// SIMATIC STEP 7 (V5.x) project zhao2017
// CPU: CPU 315-2 DP
// station: Hardware
// station: SIMATIC 300(1)
// station: P_ADR_BUS
// program: S7 Program(1)

SYMBOL_TABLE
"F1_DATA"	DB 1	DB 1
"F2_DATA"	DB 2	DB 2
"DI/DO测试程序"	FC 31	FC 31
"AI/AO测试程序"	FC 32	FC 32
"端子控制"	FC 41	FC 41
"PPO1通讯子程序"	FC 60	FC 60
"单机启停控制"	FC 71	FC 71
"加减速子程序"	FC 72	FC 72
"同步逻辑程序"	FC 81	FC 81
"单机速度程序"	FC 82	FC 82
"同步速度程序"	FC 83	FC 83
"显示与通讯程序"	FC 84	FC 84
"S1_run"	I 0.0	BOOL	// M150.0
"S1_stop"	I 0.1	BOOL	// M150.1
"S1_inc"	I 0.2	BOOL	// M150.2
"S1_dec"	I 0.3	BOOL	// M150.3
"S4_run"	I 1.4	BOOL	// M150.6
"S4_stop"	I 1.5	BOOL	// M150.7
"S4_inc"	I 1.6	BOOL	// M151.0
"S4_dec"	I 1.7	BOOL	// M151.1
"S5_run"	I 4.0	BOOL	// M151.4
"S5_stop"	I 4.1	BOOL	// M151.5
"F1"	I 6.0	BOOL	// M151.6
"F2"	I 6.1	BOOL	// M151.7
"zeroadj"	I 6.6	BOOL
"maxadj"	I 6.7	BOOL
"pulse"	M 20.0	BOOL
"T1S"	M 20.1	BOOL
"S1_running"	M 70.0	BOOL
"S4_running"	M 70.1	BOOL
"S1_Run_Mode"	M 70.2	BOOL
"S4_Run_Mode"	M 70.5	BOOL
"S1_P1"	M 80.0	BOOL
"S1_P2"	M 80.1	BOOL
"S1_P3"	M 80.2	BOOL
"S1_P4"	M 80.3	BOOL
"S1_P5"	M 80.4	BOOL
"S1_P6"	M 80.5	BOOL
"S1_P7"	M 80.6	BOOL
"S4_P1"	M 81.0	BOOL
"S4_P2"	M 81.1	BOOL
"S4_P3"	M 81.2	BOOL
"S4_P4"	M 81.3	BOOL
"S4_P5"	M 81.4	BOOL
"S4_P6"	M 81.5	BOOL
"S4_P7"	M 81.6	BOOL
"S4_P8"	M 81.7	BOOL
"S1_P8"	M 82.0	BOOL
"S1_stoped"	M 82.2	BOOL
"S4_stoped"	M 82.3	BOOL
"S1_running_order"	M 83.0	BOOL
"S4_running_order"	M 83.1	BOOL
"T50ms"	M 200.0	BOOL
"S1_running_p"	M 200.1	BOOL
"T 50MS"	M 200.2	BOOL
"S4_running_p"	M 200.3	BOOL
"S1_speed"	PQW 304	WORD
"S5_speed"	PQW 308	WORD
"S4_speed"	PQW 310	WORD
"S5_1speed"	PQW 320	WORD
"S1_run_lamp"	Q 8.0	BOOL	// M150.4
"S1_stop_lamp"	Q 8.1	BOOL	// M150.5
"S4_run_lamp"	Q 8.6	BOOL	// M151.2
"S4_stop_lamp"	Q 8.7	BOOL	// M151.3
"DPRD_DAT"	SFC 14	SFC 14	// Read Consistent Data of a Standard DP Slave
"DPWR_DAT"	SFC 15	SFC 15	// Write Consistent Data to a Standard DP Slave
END_SYMBOL_TABLE

FUNCTION "DI/DO测试程序" : VOID	// FC 31
VERSION : 0.1
BEGIN
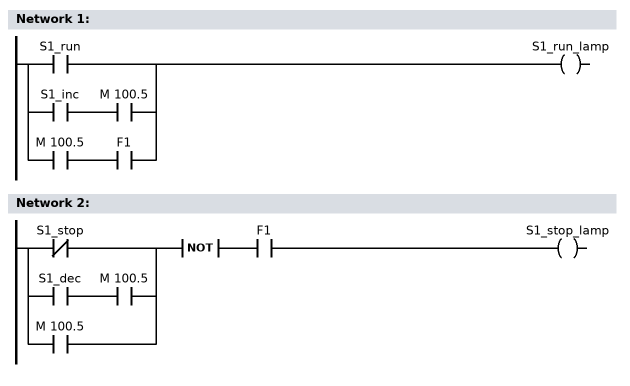
NETWORK
TITLE =
      O     "S1_run";
      O;
      A     "S1_inc";
      A     M 100.5;
      O;
      A     M 100.5;
      A     "F1";
      =     "S1_run_lamp";
NETWORK
TITLE =
      ON    "S1_stop";
      O;
      A     "S1_dec";
      A     M 100.5;
      O;
      A     M 100.5;
      NOT;
      A     "F1";
      =     "S1_stop_lamp";
END_FUNCTION

FUNCTION "AI/AO测试程序" : VOID	// FC 32
VERSION : 0.1
BEGIN
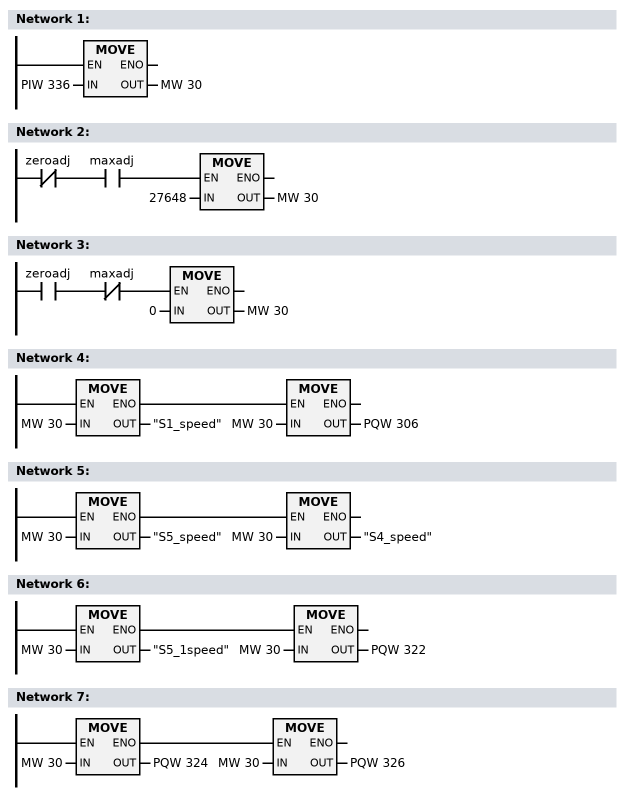
NETWORK
TITLE =
      L     PIW 336;
      T     MW 30;
      NOP   0;
NETWORK
TITLE =
      AN    "zeroadj";
      A     "maxadj";
      JNB   _001;
      L     27648;
      T     MW 30;
_001: NOP   0;
NETWORK
TITLE =
      A     "zeroadj";
      AN    "maxadj";
      JNB   _002;
      L     0;
      T     MW 30;
_002: NOP   0;
NETWORK
TITLE =
      A(;
      L     MW 30;
      T     "S1_speed";
      SET;
      SAVE;
      CLR;
      A     BR;
      );
      JNB   _003;
      L     MW 30;
      T     PQW 306;
_003: NOP   0;
NETWORK
TITLE =
      A(;
      L     MW 30;
      T     "S5_speed";
      SET;
      SAVE;
      CLR;
      A     BR;
      );
      JNB   _004;
      L     MW 30;
      T     "S4_speed";
_004: NOP   0;
NETWORK
TITLE =
      A(;
      L     MW 30;
      T     "S5_1speed";
      SET;
      SAVE;
      CLR;
      A     BR;
      );
      JNB   _005;
      L     MW 30;
      T     PQW 322;
_005: NOP   0;
NETWORK
TITLE =
      A(;
      L     MW 30;
      T     PQW 324;
      SET;
      SAVE;
      CLR;
      A     BR;
      );
      JNB   _006;
      L     MW 30;
      T     PQW 326;
_006: NOP   0;
NETWORK
TITLE =
END_FUNCTION

FUNCTION "端子控制" : VOID	// FC 41
VERSION : 0.1
BEGIN
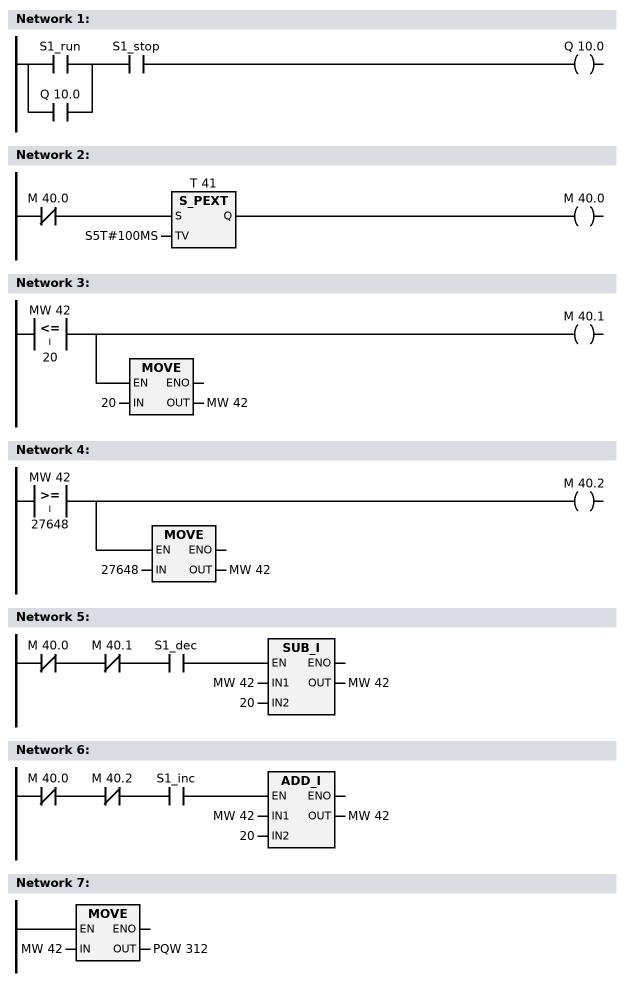
NETWORK
TITLE =
      A(;
      O     "S1_run";
      O     Q 10.0;
      );
      A     "S1_stop";
      =     Q 10.0;
NETWORK
TITLE =
      AN    M 40.0;
      L     S5T#100MS;
      SE    T 41;
      NOP   0;
      NOP   0;
      NOP   0;
      A     T 41;
      =     M 40.0;
NETWORK
TITLE =
      L     MW 42;
      L     20;
      <=I;
      =     L 0.0;
      A     L 0.0;
      BLD   102;
      =     M 40.1;
      A     L 0.0;
      JNB   _001;
      L     20;
      T     MW 42;
_001: NOP   0;
NETWORK
TITLE =
      L     MW 42;
      L     27648;
      >=I;
      =     L 0.0;
      A     L 0.0;
      BLD   102;
      =     M 40.2;
      A     L 0.0;
      JNB   _002;
      L     27648;
      T     MW 42;
_002: NOP   0;
NETWORK
TITLE =
      AN    M 40.0;
      AN    M 40.1;
      A     "S1_dec";
      JNB   _003;
      L     MW 42;
      L     20;
      -I;
      T     MW 42;
_003: NOP   0;
NETWORK
TITLE =
      AN    M 40.0;
      AN    M 40.2;
      A     "S1_inc";
      JNB   _004;
      L     MW 42;
      L     20;
      +I;
      T     MW 42;
_004: NOP   0;
NETWORK
TITLE =
      L     MW 42;
      T     PQW 312;
      NOP   0;
NETWORK
TITLE =
END_FUNCTION

FUNCTION "PPO1通讯子程序" : VOID	// FC 60
VERSION : 0.1
VAR_INPUT
  pkw1 : WORD ;
  pkw2 : WORD ;
  pkw3 : WORD ;
  pkw4 : WORD ;
  pzd1 : WORD ;
  pzd2 : INT ;
  pkw_I_addr : WORD ;
  pkw_Q_addr : WORD ;
  pzd_I_addr : WORD ;
  pzd_Q_addr : WORD ;
END_VAR
VAR_OUTPUT
  pkw1_ret : WORD ;
  pkw2_ret : WORD ;
  pkw3_ret : WORD ;
  pkw4_ret : WORD ;
  pzd1_ret : WORD ;
  pzd2_ret : WORD ;
  err : BOOL ;
END_VAR
VAR_TEMP
  pkw : STRUCT
   w1 : WORD ;
   w2 : WORD ;
   w3 : WORD ;
   w4 : WORD ;
  END_STRUCT ;
  pzd : STRUCT
   w1 : WORD ;
   w2 : WORD ;
  END_STRUCT ;
  pkw_RD : STRUCT
   w1 : WORD ;
   w2 : WORD ;
   w3 : WORD ;
   w4 : WORD ;
  END_STRUCT ;
  pzd_RD : STRUCT
   w1 : WORD ;
   w2 : WORD ;
  END_STRUCT ;
  tt : STRUCT
   w1 : INT ;
   w2 : INT ;
   w3 : INT ;
   w4 : INT ;
  END_STRUCT ;
END_VAR
BEGIN
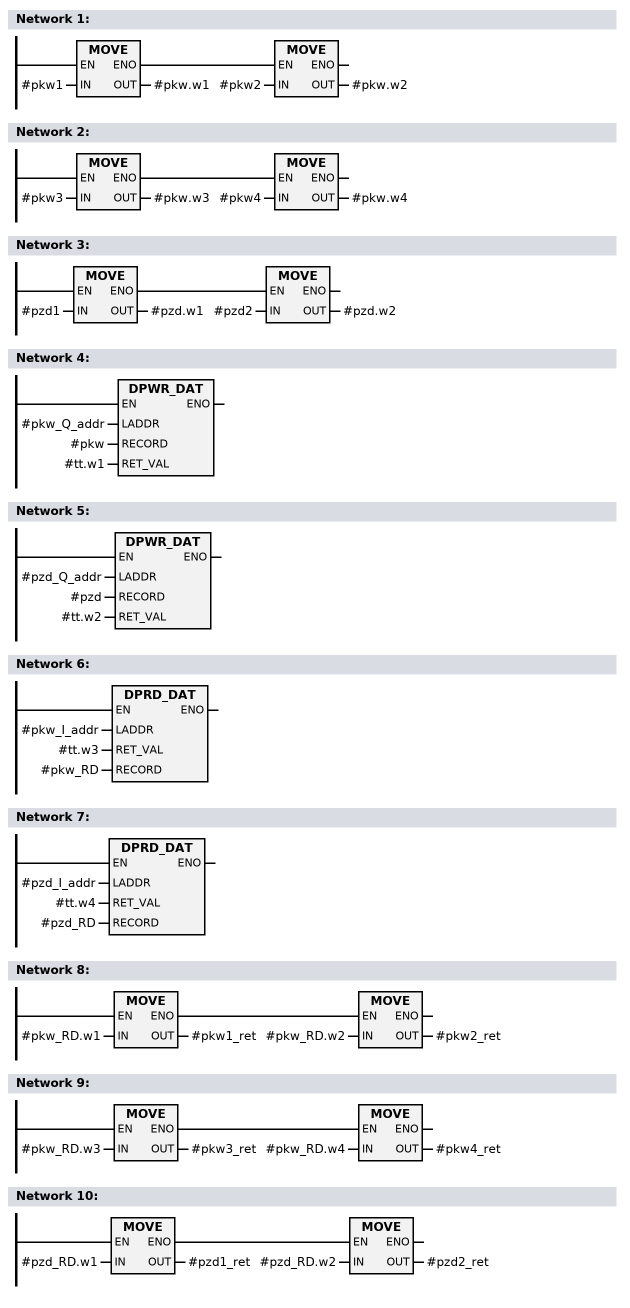
NETWORK
TITLE =
//将pkw1、pkw2数据放入变量组
      A(;
      L     #pkw1;
      T     #pkw.w1;
      SET;
      SAVE;
      CLR;
      A     BR;
      );
      JNB   _001;
      L     #pkw2;
      T     #pkw.w2;
_001: NOP   0;
NETWORK
TITLE =
//将pkw3、pkw4数据放入变量组
      A(;
      L     #pkw3;
      T     #pkw.w3;
      SET;
      SAVE;
      CLR;
      A     BR;
      );
      JNB   _002;
      L     #pkw4;
      T     #pkw.w4;
_002: NOP   0;
NETWORK
TITLE =
//将pzd数据放入变量组
      A(;
      L     #pzd1;
      T     #pzd.w1;
      SET;
      SAVE;
      CLR;
      A     BR;
      );
      JNB   _003;
      L     #pzd2;
      T     #pzd.w2;
_003: NOP   0;
NETWORK
TITLE =
//将pkw数据输出
      CALL  "DPWR_DAT" (
           LADDR                    := #pkw_Q_addr,
           RECORD                   := #pkw,
           RET_VAL                  := #tt.w1);
      NOP   0;
NETWORK
TITLE =
//将pzd数据输出
      CALL  "DPWR_DAT" (
           LADDR                    := #pzd_Q_addr,
           RECORD                   := #pzd,
           RET_VAL                  := #tt.w2);
      NOP   0;
NETWORK
TITLE =
//将pkw响应数据读入
      CALL  "DPRD_DAT" (
           LADDR                    := #pkw_I_addr,
           RET_VAL                  := #tt.w3,
           RECORD                   := #pkw_RD);
      NOP   0;
NETWORK
TITLE =
//将pzd响应数据读入
      CALL  "DPRD_DAT" (
           LADDR                    := #pzd_I_addr,
           RET_VAL                  := #tt.w4,
           RECORD                   := #pzd_RD);
      NOP   0;
NETWORK
TITLE =
//把读入的数据放入PKW响应数据区相应位置
      A(;
      L     #pkw_RD.w1;
      T     #pkw1_ret;
      SET;
      SAVE;
      CLR;
      A     BR;
      );
      JNB   _004;
      L     #pkw_RD.w2;
      T     #pkw2_ret;
_004: NOP   0;
NETWORK
TITLE =
//把读入的数据放入PKW响应数据区相应位置
      A(;
      L     #pkw_RD.w3;
      T     #pkw3_ret;
      SET;
      SAVE;
      CLR;
      A     BR;
      );
      JNB   _005;
      L     #pkw_RD.w4;
      T     #pkw4_ret;
_005: NOP   0;
NETWORK
TITLE =
//把读入的数据放入PZD响应数据区相应位置
      A(;
      L     #pzd_RD.w1;
      T     #pzd1_ret;
      SET;
      SAVE;
      CLR;
      A     BR;
      );
      JNB   _006;
      L     #pzd_RD.w2;
      T     #pzd2_ret;
_006: NOP   0;
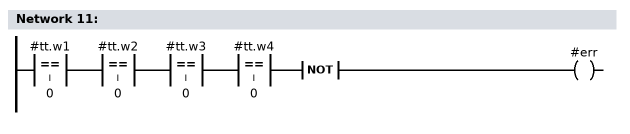
NETWORK
TITLE =
      A(;
      L     #tt.w1;
      L     0;
      ==I;
      );
      A(;
      L     #tt.w2;
      L     0;
      ==I;
      );
      A(;
      L     #tt.w3;
      L     0;
      ==I;
      );
      A(;
      L     #tt.w4;
      L     0;
      ==I;
      );
      NOT;
      =     #err;
END_FUNCTION

FUNCTION "单机启停控制" : VOID	// FC 71
VERSION : 0.1
BEGIN
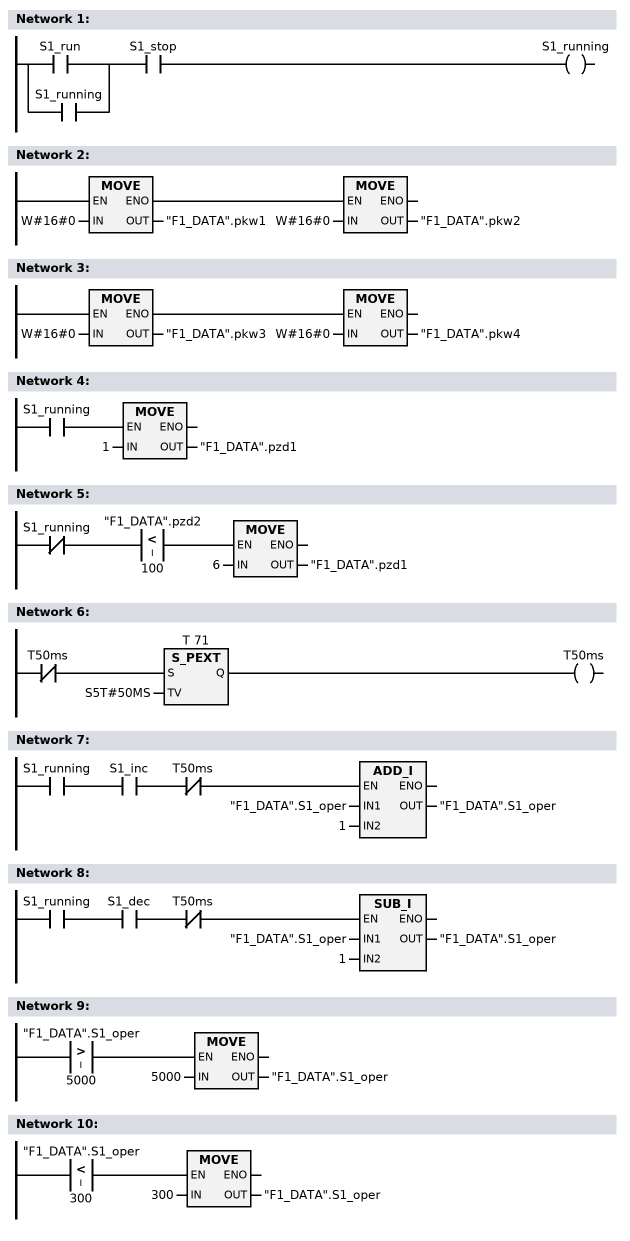
NETWORK
TITLE =
      A(;
      O     "S1_run";
      O     "S1_running";
      );
      A     "S1_stop";
      =     "S1_running";
NETWORK
TITLE =
      A(;
      L     W#16#0;
      T     "F1_DATA".pkw1;
      SET;
      SAVE;
      CLR;
      A     BR;
      );
      JNB   _001;
      L     W#16#0;
      T     "F1_DATA".pkw2;
_001: NOP   0;
NETWORK
TITLE =
      A(;
      L     W#16#0;
      T     "F1_DATA".pkw3;
      SET;
      SAVE;
      CLR;
      A     BR;
      );
      JNB   _002;
      L     W#16#0;
      T     "F1_DATA".pkw4;
_002: NOP   0;
NETWORK
TITLE =
      A     "S1_running";
      JNB   _003;
      L     1;
      T     "F1_DATA".pzd1;
_003: NOP   0;
NETWORK
TITLE =
      AN    "S1_running";
      A(;
      L     "F1_DATA".pzd2;
      L     100;
      <I;
      );
      JNB   _004;
      L     6;
      T     "F1_DATA".pzd1;
_004: NOP   0;
NETWORK
TITLE =
      AN    "T50ms";
      L     S5T#50MS;
      SE    T 71;
      NOP   0;
      NOP   0;
      NOP   0;
      A     T 71;
      =     "T50ms";
NETWORK
TITLE =
      A     "S1_running";
      A     "S1_inc";
      AN    "T50ms";
      JNB   _005;
      L     "F1_DATA".S1_oper;
      L     1;
      +I;
      T     "F1_DATA".S1_oper;
_005: NOP   0;
NETWORK
TITLE =
      A     "S1_running";
      A     "S1_dec";
      AN    "T50ms";
      JNB   _006;
      L     "F1_DATA".S1_oper;
      L     1;
      -I;
      T     "F1_DATA".S1_oper;
_006: NOP   0;
NETWORK
TITLE =
      A(;
      L     "F1_DATA".S1_oper;
      L     5000;
      >I;
      );
      JNB   _007;
      L     5000;
      T     "F1_DATA".S1_oper;
_007: NOP   0;
NETWORK
TITLE =
      A(;
      L     "F1_DATA".S1_oper;
      L     300;
      <I;
      );
      JNB   _008;
      L     300;
      T     "F1_DATA".S1_oper;
_008: NOP   0;
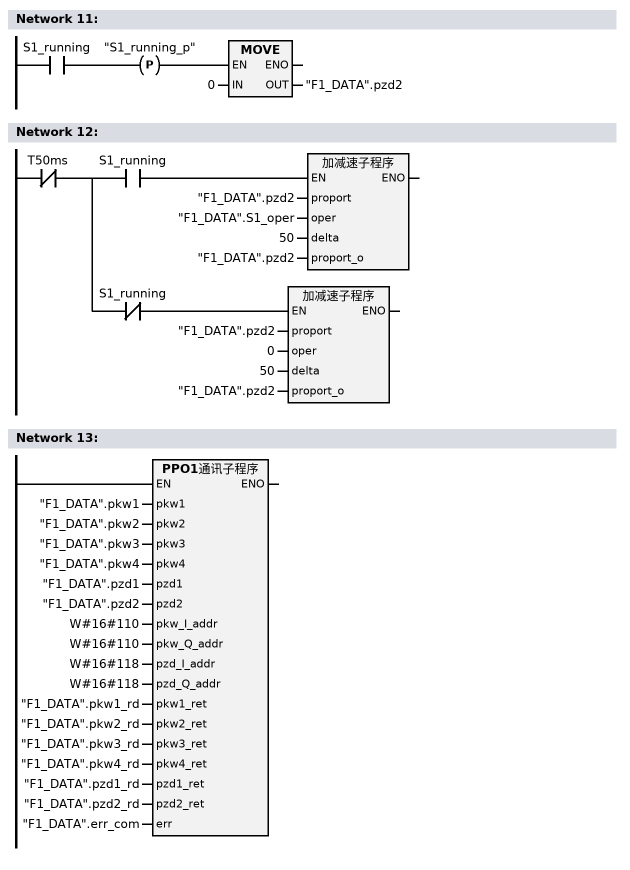
NETWORK
TITLE =
      A     "S1_running";
      FP    "S1_running_p";
      JNB   _009;
      L     0;
      T     "F1_DATA".pzd2;
_009: NOP   0;
NETWORK
TITLE =
      AN    "T50ms";
      =     L 0.0;
      A     L 0.0;
      A     "S1_running";
      JNB   _00a;
      CALL  "加减速子程序" (
           proport                  := "F1_DATA".pzd2,
           oper                     := "F1_DATA".S1_oper,
           delta                    := 50,
           proport_o                := "F1_DATA".pzd2);
_00a: NOP   0;
      A     L 0.0;
      AN    "S1_running";
      JNB   _00b;
      CALL  "加减速子程序" (
           proport                  := "F1_DATA".pzd2,
           oper                     := 0,
           delta                    := 50,
           proport_o                := "F1_DATA".pzd2);
_00b: NOP   0;
NETWORK
TITLE =
      CALL  "PPO1通讯子程序" (
           pkw1                     := "F1_DATA".pkw1,
           pkw2                     := "F1_DATA".pkw2,
           pkw3                     := "F1_DATA".pkw3,
           pkw4                     := "F1_DATA".pkw4,
           pzd1                     := "F1_DATA".pzd1,
           pzd2                     := "F1_DATA".pzd2,
           pkw_I_addr               := W#16#110,
           pkw_Q_addr               := W#16#110,
           pzd_I_addr               := W#16#118,
           pzd_Q_addr               := W#16#118,
           pkw1_ret                 := "F1_DATA".pkw1_rd,
           pkw2_ret                 := "F1_DATA".pkw2_rd,
           pkw3_ret                 := "F1_DATA".pkw3_rd,
           pkw4_ret                 := "F1_DATA".pkw4_rd,
           pzd1_ret                 := "F1_DATA".pzd1_rd,
           pzd2_ret                 := "F1_DATA".pzd2_rd,
           err                      := "F1_DATA".err_com);
      NOP   0;
END_FUNCTION

FUNCTION "加减速子程序" : VOID	// FC 72
VERSION : 0.1
VAR_INPUT
  proport : INT ;
  oper : INT ;
  delta : INT ;
END_VAR
VAR_OUTPUT
  proport_o : INT ;
END_VAR
VAR_TEMP
  temp1 : BOOL ;
  temp2 : INT ;
END_VAR
BEGIN
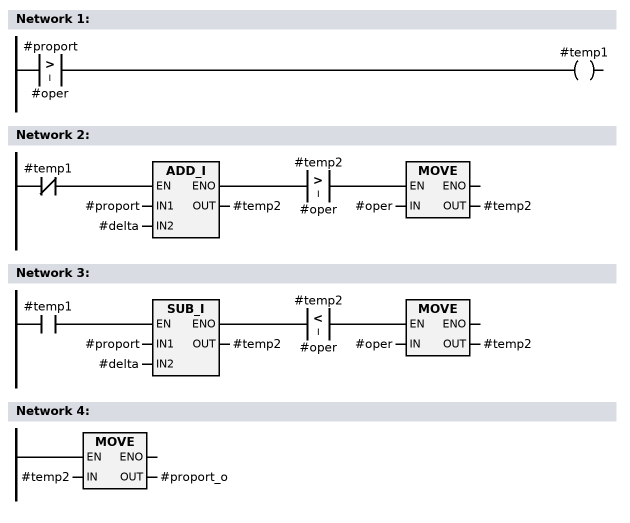
NETWORK
TITLE =
      L     #proport;
      L     #oper;
      >I;
      =     #temp1;
NETWORK
TITLE =
      A(;
      AN    #temp1;
      JNB   _001;
      L     #proport;
      L     #delta;
      +I;
      T     #temp2;
      AN    OV;
      SAVE;
      CLR;
_001: A     BR;
      );
      A(;
      L     #temp2;
      L     #oper;
      >I;
      );
      JNB   _002;
      L     #oper;
      T     #temp2;
_002: NOP   0;
NETWORK
TITLE =
      A(;
      A     #temp1;
      JNB   _003;
      L     #proport;
      L     #delta;
      -I;
      T     #temp2;
      AN    OV;
      SAVE;
      CLR;
_003: A     BR;
      );
      A(;
      L     #temp2;
      L     #oper;
      <I;
      );
      JNB   _004;
      L     #oper;
      T     #temp2;
_004: NOP   0;
NETWORK
TITLE =
      L     #temp2;
      T     #proport_o;
      NOP   0;
END_FUNCTION

FUNCTION "同步逻辑程序" : VOID	// FC 81
VERSION : 0.1
BEGIN
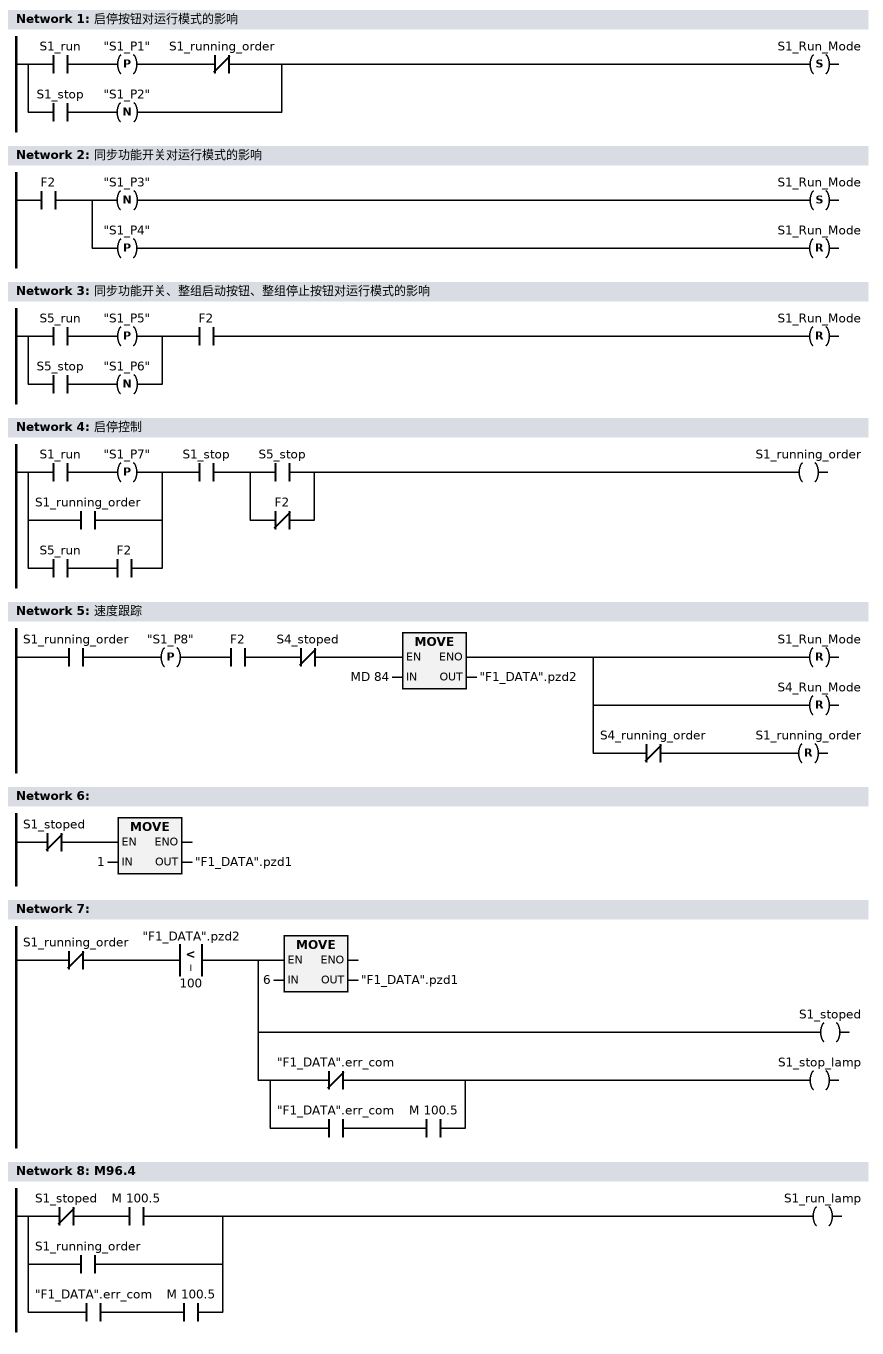
NETWORK
TITLE = 启停按钮对运行模式的影响
//Run_Mode=1表示单机运行，Run_Mode=0表示同步运行
      A     "S1_run";
      FP    "S1_P1";
      AN    "S1_running_order";
      O(;
      A     "S1_stop";
      FN    "S1_P2";
      );
      S     "S1_Run_Mode";
NETWORK
TITLE = 同步功能开关对运行模式的影响
//Run_Mode=1表示单机运行，Run_Mode=0表示同步运行
      A     "F2";
      =     L 0.0;
      A     L 0.0;
      FN    "S1_P3";
      S     "S1_Run_Mode";
      A     L 0.0;
      FP    "S1_P4";
      R     "S1_Run_Mode";
NETWORK
TITLE = 同步功能开关、整组启动按钮、整组停止按钮对运行模式的影响
//Run_Mode=1表示单机运行，Run_Mode=0表示同步运行
//“S3启动”（I1.0）为整组启动按钮，“S3停止”（I1.1）为整组停止按钮。
      A(;
      A     "S5_run";
      FP    "S1_P5";
      O(;
      A     "S5_stop";
      FN    "S1_P6";
      );
      );
      A     "F2";
      R     "S1_Run_Mode";
NETWORK
TITLE = 启停控制
//“F2”（I6.1）为同步功能开关，即I6.1=0时，两台变频器单机运行，I6.1=1时，两台变频
//器同步运行
      A(;
      A     "S1_run";
      FP    "S1_P7";
      O     "S1_running_order";
      O;
      A     "S5_run";
      A     "F2";
      );
      A     "S1_stop";
      A(;
      O     "S5_stop";
      ON    "F2";
      );
      =     "S1_running_order";
NETWORK
TITLE = 速度跟踪
//Run_Mode=1表示单机运行，Run_Mode=0表示同步运行
      A     "S1_running_order";
      FP    "S1_P8";
      A     "F2";
      AN    "S4_stoped";
      JNB   _001;
      L     MD 84;
      T     "F1_DATA".pzd2;
      SET;
      SAVE;
      CLR;
_001: A     BR;
      =     L 0.0;
      A     L 0.0;
      BLD   102;
      R     "S1_Run_Mode";
      A     L 0.0;
      BLD   102;
      R     "S4_Run_Mode";
      A     L 0.0;
      AN    "S4_running_order";
      R     "S1_running_order";
NETWORK
TITLE =
      AN    "S1_stoped";
      JNB   _002;
      L     1;
      T     "F1_DATA".pzd1;
_002: NOP   0;
NETWORK
TITLE =
      AN    "S1_running_order";
      A(;
      L     "F1_DATA".pzd2;
      L     100;
      <I;
      );
      =     L 0.0;
      A     L 0.0;
      JNB   _003;
      L     6;
      T     "F1_DATA".pzd1;
_003: NOP   0;
      A     L 0.0;
      BLD   102;
      =     "S1_stoped";
      A     L 0.0;
      A(;
      ON    "F1_DATA".err_com;
      O;
      A     "F1_DATA".err_com;
      A     M 100.5;
      );
      =     "S1_stop_lamp";
NETWORK
TITLE = M96.4
      AN    "S1_stoped";
      A     M 100.5;
      O     "S1_running_order";
      O;
      A     "F1_DATA".err_com;
      A     M 100.5;
      =     "S1_run_lamp";
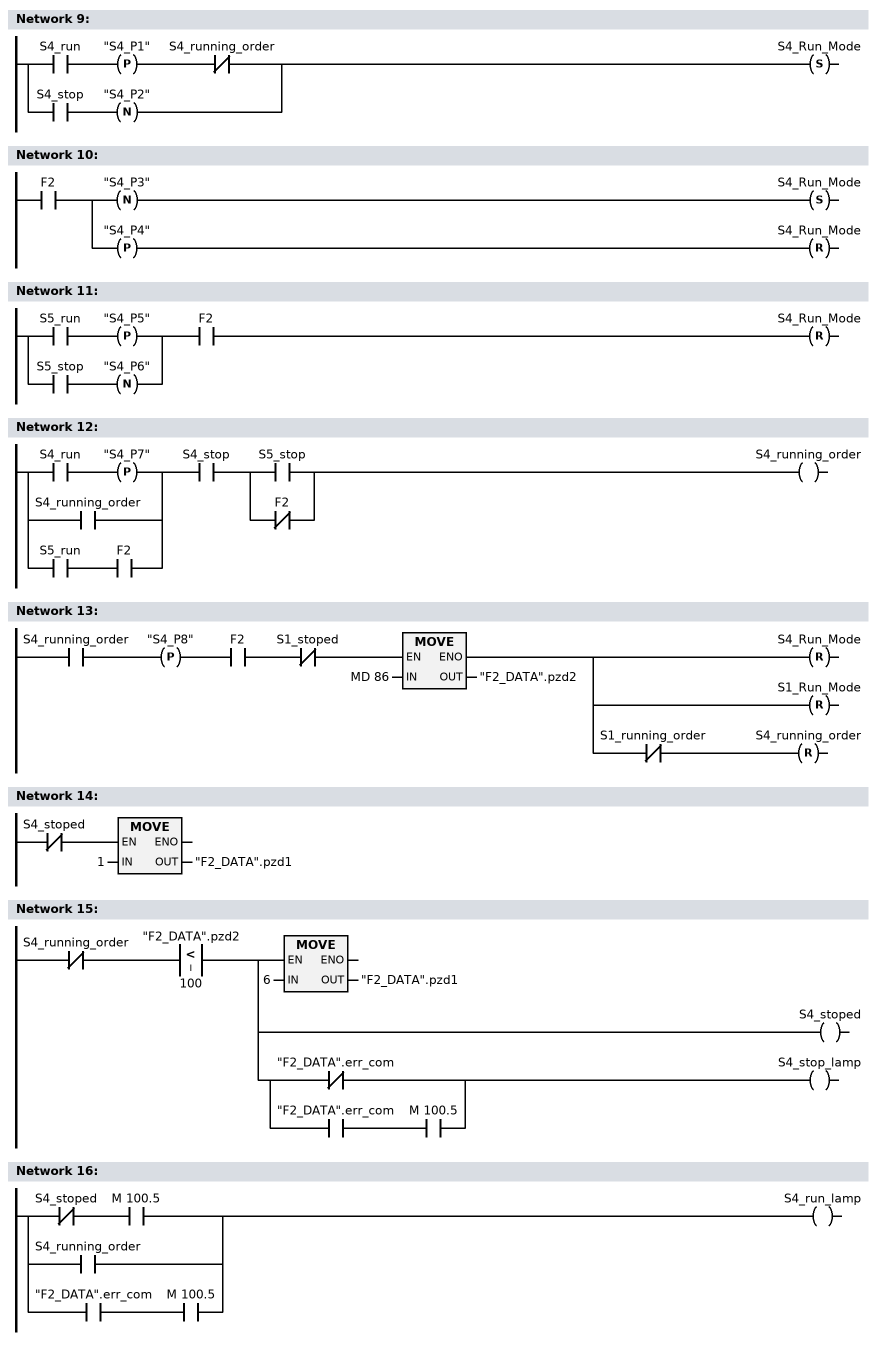
NETWORK
TITLE =
      A     "S4_run";
      FP    "S4_P1";
      AN    "S4_running_order";
      O(;
      A     "S4_stop";
      FN    "S4_P2";
      );
      S     "S4_Run_Mode";
NETWORK
TITLE =
      A     "F2";
      =     L 0.0;
      A     L 0.0;
      FN    "S4_P3";
      S     "S4_Run_Mode";
      A     L 0.0;
      FP    "S4_P4";
      R     "S4_Run_Mode";
NETWORK
TITLE =
      A(;
      A     "S5_run";
      FP    "S4_P5";
      O(;
      A     "S5_stop";
      FN    "S4_P6";
      );
      );
      A     "F2";
      R     "S4_Run_Mode";
NETWORK
TITLE =
      A(;
      A     "S4_run";
      FP    "S4_P7";
      O     "S4_running_order";
      O;
      A     "S5_run";
      A     "F2";
      );
      A     "S4_stop";
      A(;
      O     "S5_stop";
      ON    "F2";
      );
      =     "S4_running_order";
NETWORK
TITLE =
      A     "S4_running_order";
      FP    "S4_P8";
      A     "F2";
      AN    "S1_stoped";
      JNB   _004;
      L     MD 86;
      T     "F2_DATA".pzd2;
      SET;
      SAVE;
      CLR;
_004: A     BR;
      =     L 0.0;
      A     L 0.0;
      BLD   102;
      R     "S4_Run_Mode";
      A     L 0.0;
      BLD   102;
      R     "S1_Run_Mode";
      A     L 0.0;
      AN    "S1_running_order";
      R     "S4_running_order";
NETWORK
TITLE =
      AN    "S4_stoped";
      JNB   _005;
      L     1;
      T     "F2_DATA".pzd1;
_005: NOP   0;
NETWORK
TITLE =
      AN    "S4_running_order";
      A(;
      L     "F2_DATA".pzd2;
      L     100;
      <I;
      );
      =     L 0.0;
      A     L 0.0;
      JNB   _006;
      L     6;
      T     "F2_DATA".pzd1;
_006: NOP   0;
      A     L 0.0;
      BLD   102;
      =     "S4_stoped";
      A     L 0.0;
      A(;
      ON    "F2_DATA".err_com;
      O;
      A     "F2_DATA".err_com;
      A     M 100.5;
      );
      =     "S4_stop_lamp";
NETWORK
TITLE =
      AN    "S4_stoped";
      A     M 100.5;
      O     "S4_running_order";
      O;
      A     "F2_DATA".err_com;
      A     M 100.5;
      =     "S4_run_lamp";
END_FUNCTION

FUNCTION "单机速度程序" : VOID	// FC 82
VERSION : 0.1
VAR_TEMP
  S1_di_su : INT ;
  S2_di_su : INT ;
END_VAR
BEGIN
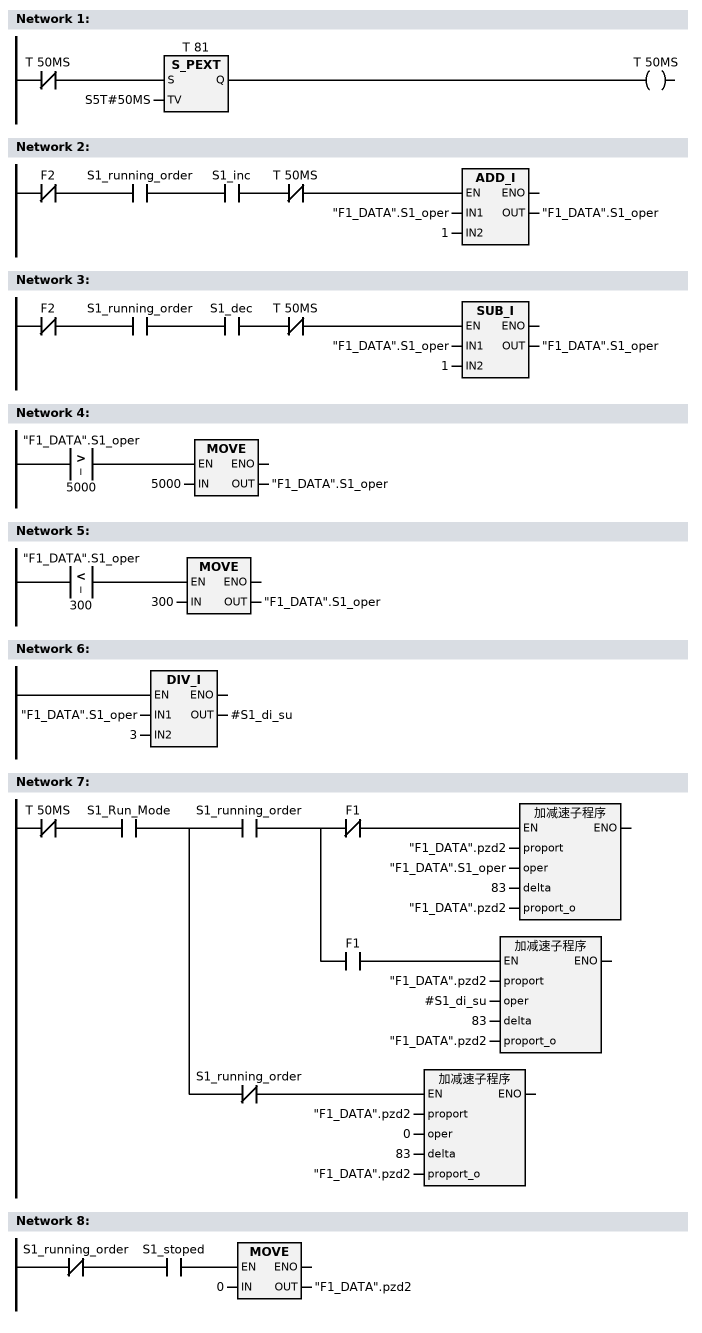
NETWORK
TITLE =
      AN    "T 50MS";
      L     S5T#50MS;
      SE    T 81;
      NOP   0;
      NOP   0;
      NOP   0;
      A     T 81;
      =     "T 50MS";
NETWORK
TITLE =
      AN    "F2";
      A     "S1_running_order";
      A     "S1_inc";
      AN    "T 50MS";
      JNB   _001;
      L     "F1_DATA".S1_oper;
      L     1;
      +I;
      T     "F1_DATA".S1_oper;
_001: NOP   0;
NETWORK
TITLE =
      AN    "F2";
      A     "S1_running_order";
      A     "S1_dec";
      AN    "T 50MS";
      JNB   _002;
      L     "F1_DATA".S1_oper;
      L     1;
      -I;
      T     "F1_DATA".S1_oper;
_002: NOP   0;
NETWORK
TITLE =
      A(;
      L     "F1_DATA".S1_oper;
      L     5000;
      >I;
      );
      JNB   _003;
      L     5000;
      T     "F1_DATA".S1_oper;
_003: NOP   0;
NETWORK
TITLE =
      A(;
      L     "F1_DATA".S1_oper;
      L     300;
      <I;
      );
      JNB   _004;
      L     300;
      T     "F1_DATA".S1_oper;
_004: NOP   0;
NETWORK
TITLE =
      L     "F1_DATA".S1_oper;
      L     3;
      /I;
      T     #S1_di_su;
      NOP   0;
NETWORK
TITLE =
      AN    "T 50MS";
      A     "S1_Run_Mode";
      =     L 4.0;
      A     L 4.0;
      A     "S1_running_order";
      =     L 4.1;
      A     L 4.1;
      AN    "F1";
      JNB   _005;
      CALL  "加减速子程序" (
           proport                  := "F1_DATA".pzd2,
           oper                     := "F1_DATA".S1_oper,
           delta                    := 83,
           proport_o                := "F1_DATA".pzd2);
_005: NOP   0;
      A     L 4.1;
      A     "F1";
      JNB   _006;
      CALL  "加减速子程序" (
           proport                  := "F1_DATA".pzd2,
           oper                     := #S1_di_su,
           delta                    := 83,
           proport_o                := "F1_DATA".pzd2);
_006: NOP   0;
      A     L 4.0;
      AN    "S1_running_order";
      JNB   _007;
      CALL  "加减速子程序" (
           proport                  := "F1_DATA".pzd2,
           oper                     := 0,
           delta                    := 83,
           proport_o                := "F1_DATA".pzd2);
_007: NOP   0;
NETWORK
TITLE =
      AN    "S1_running_order";
      A     "S1_stoped";
      JNB   _008;
      L     0;
      T     "F1_DATA".pzd2;
_008: NOP   0;
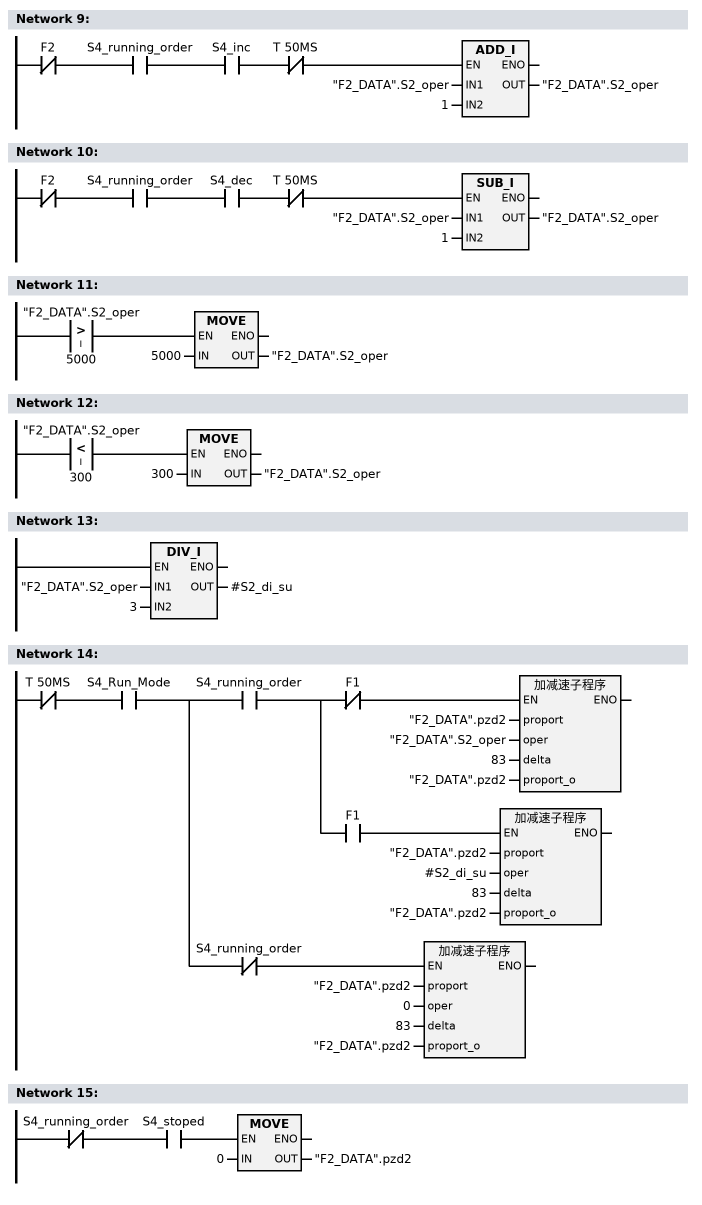
NETWORK
TITLE =
      AN    "F2";
      A     "S4_running_order";
      A     "S4_inc";
      AN    "T 50MS";
      JNB   _009;
      L     "F2_DATA".S2_oper;
      L     1;
      +I;
      T     "F2_DATA".S2_oper;
_009: NOP   0;
NETWORK
TITLE =
      AN    "F2";
      A     "S4_running_order";
      A     "S4_dec";
      AN    "T 50MS";
      JNB   _00a;
      L     "F2_DATA".S2_oper;
      L     1;
      -I;
      T     "F2_DATA".S2_oper;
_00a: NOP   0;
NETWORK
TITLE =
      A(;
      L     "F2_DATA".S2_oper;
      L     5000;
      >I;
      );
      JNB   _00b;
      L     5000;
      T     "F2_DATA".S2_oper;
_00b: NOP   0;
NETWORK
TITLE =
      A(;
      L     "F2_DATA".S2_oper;
      L     300;
      <I;
      );
      JNB   _00c;
      L     300;
      T     "F2_DATA".S2_oper;
_00c: NOP   0;
NETWORK
TITLE =
      L     "F2_DATA".S2_oper;
      L     3;
      /I;
      T     #S2_di_su;
      NOP   0;
NETWORK
TITLE =
      AN    "T 50MS";
      A     "S4_Run_Mode";
      =     L 4.0;
      A     L 4.0;
      A     "S4_running_order";
      =     L 4.1;
      A     L 4.1;
      AN    "F1";
      JNB   _00d;
      CALL  "加减速子程序" (
           proport                  := "F2_DATA".pzd2,
           oper                     := "F2_DATA".S2_oper,
           delta                    := 83,
           proport_o                := "F2_DATA".pzd2);
_00d: NOP   0;
      A     L 4.1;
      A     "F1";
      JNB   _00e;
      CALL  "加减速子程序" (
           proport                  := "F2_DATA".pzd2,
           oper                     := #S2_di_su,
           delta                    := 83,
           proport_o                := "F2_DATA".pzd2);
_00e: NOP   0;
      A     L 4.0;
      AN    "S4_running_order";
      JNB   _00f;
      CALL  "加减速子程序" (
           proport                  := "F2_DATA".pzd2,
           oper                     := 0,
           delta                    := 83,
           proport_o                := "F2_DATA".pzd2);
_00f: NOP   0;
NETWORK
TITLE =
      AN    "S4_running_order";
      A     "S4_stoped";
      JNB   _010;
      L     0;
      T     "F2_DATA".pzd2;
_010: NOP   0;
END_FUNCTION

FUNCTION "同步速度程序" : VOID	// FC 83
VERSION : 0.1
VAR_TEMP
  TEMP0 : DINT ;
  TEMP1 : REAL ;
  TEMP2 : DINT ;
  TEMP3 : REAL ;
  S1_di_su : INT ;
  S2_di_su : INT ;
END_VAR
BEGIN
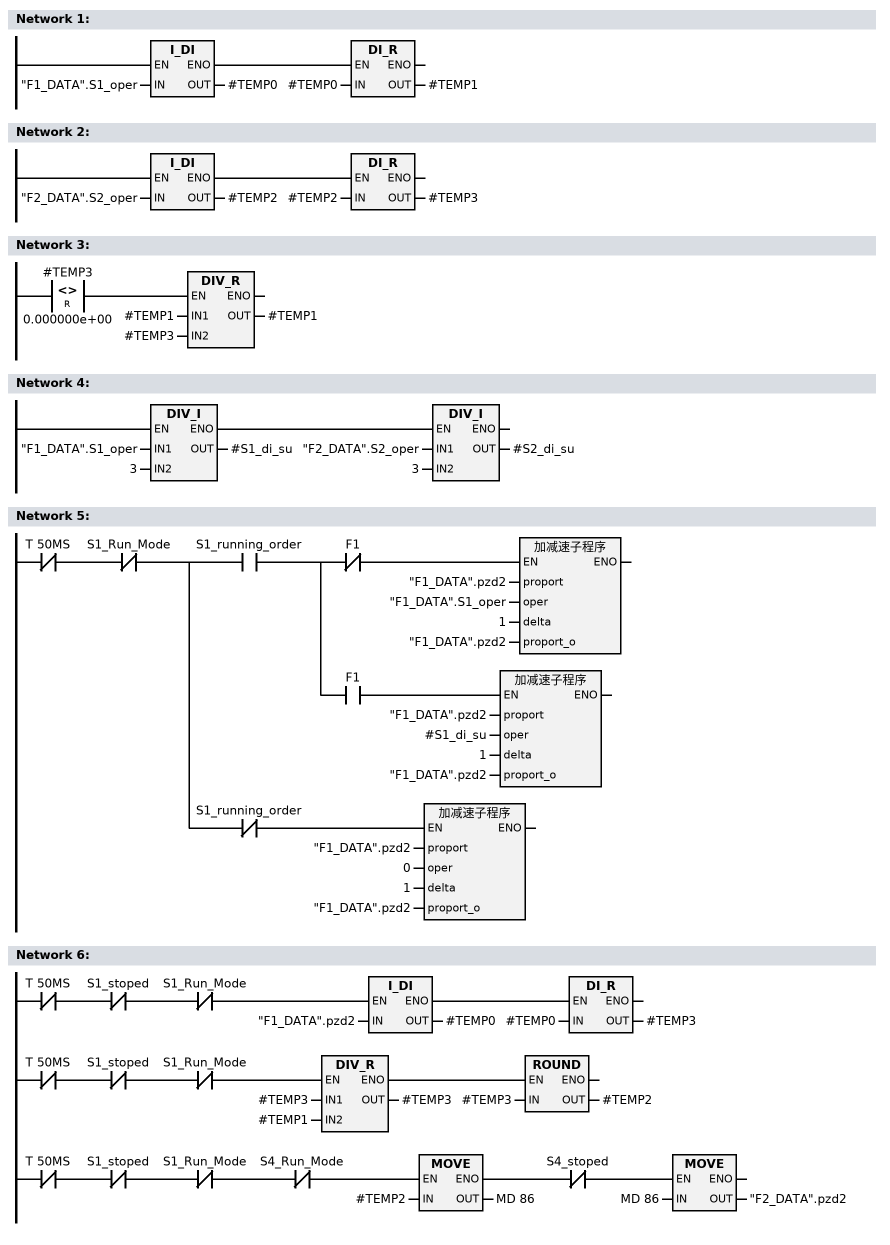
NETWORK
TITLE =
      A(;
      L     "F1_DATA".S1_oper;
      ITD;
      T     #TEMP0;
      SET;
      SAVE;
      CLR;
      A     BR;
      );
      JNB   _001;
      L     #TEMP0;
      DTR;
      T     #TEMP1;
_001: NOP   0;
NETWORK
TITLE =
      A(;
      L     "F2_DATA".S2_oper;
      ITD;
      T     #TEMP2;
      SET;
      SAVE;
      CLR;
      A     BR;
      );
      JNB   _002;
      L     #TEMP2;
      DTR;
      T     #TEMP3;
_002: NOP   0;
NETWORK
TITLE =
      A(;
      L     #TEMP3;
      L     0.000000e+00;
      <>R;
      );
      JNB   _003;
      L     #TEMP1;
      L     #TEMP3;
      /R;
      T     #TEMP1;
_003: NOP   0;
NETWORK
TITLE =
      A(;
      L     "F1_DATA".S1_oper;
      L     3;
      /I;
      T     #S1_di_su;
      AN    OV;
      SAVE;
      CLR;
      A     BR;
      );
      JNB   _004;
      L     "F2_DATA".S2_oper;
      L     3;
      /I;
      T     #S2_di_su;
_004: NOP   0;
NETWORK
TITLE =
      AN    "T 50MS";
      AN    "S1_Run_Mode";
      =     L 20.0;
      A     L 20.0;
      A     "S1_running_order";
      =     L 20.1;
      A     L 20.1;
      AN    "F1";
      JNB   _005;
      CALL  "加减速子程序" (
           proport                  := "F1_DATA".pzd2,
           oper                     := "F1_DATA".S1_oper,
           delta                    := 1,
           proport_o                := "F1_DATA".pzd2);
_005: NOP   0;
      A     L 20.1;
      A     "F1";
      JNB   _006;
      CALL  "加减速子程序" (
           proport                  := "F1_DATA".pzd2,
           oper                     := #S1_di_su,
           delta                    := 1,
           proport_o                := "F1_DATA".pzd2);
_006: NOP   0;
      A     L 20.0;
      AN    "S1_running_order";
      JNB   _007;
      CALL  "加减速子程序" (
           proport                  := "F1_DATA".pzd2,
           oper                     := 0,
           delta                    := 1,
           proport_o                := "F1_DATA".pzd2);
_007: NOP   0;
NETWORK
TITLE =
      AN    "T 50MS";
      AN    "S1_stoped";
      AN    "S1_Run_Mode";
      =     L 20.0;
      A(;
      A     L 20.0;
      JNB   _008;
      L     "F1_DATA".pzd2;
      ITD;
      T     #TEMP0;
      SET;
      SAVE;
      CLR;
_008: A     BR;
      );
      JNB   _009;
      L     #TEMP0;
      DTR;
      T     #TEMP3;
_009: NOP   0;
      A(;
      A     L 20.0;
      JNB   _00a;
      L     #TEMP3;
      L     #TEMP1;
      /R;
      T     #TEMP3;
      AN    OV;
      SAVE;
      CLR;
_00a: A     BR;
      );
      JNB   _00b;
      L     #TEMP3;
      RND;
      T     #TEMP2;
_00b: NOP   0;
      A(;
      A     L 20.0;
      AN    "S4_Run_Mode";
      JNB   _00c;
      L     #TEMP2;
      T     MD 86;
      SET;
      SAVE;
      CLR;
_00c: A     BR;
      );
      AN    "S4_stoped";
      JNB   _00d;
      L     MD 86;
      T     "F2_DATA".pzd2;
_00d: NOP   0;
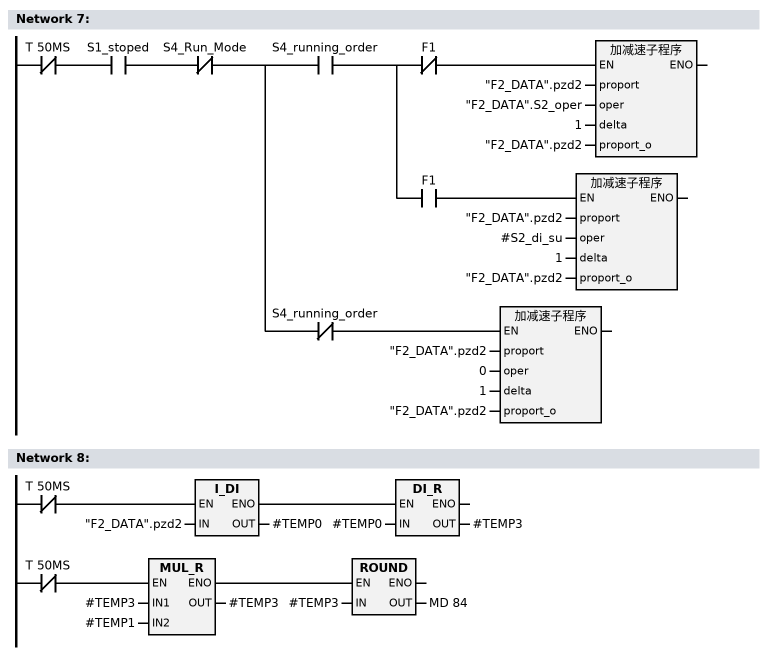
NETWORK
TITLE =
      AN    "T 50MS";
      A     "S1_stoped";
      AN    "S4_Run_Mode";
      =     L 20.0;
      A     L 20.0;
      A     "S4_running_order";
      =     L 20.1;
      A     L 20.1;
      AN    "F1";
      JNB   _00e;
      CALL  "加减速子程序" (
           proport                  := "F2_DATA".pzd2,
           oper                     := "F2_DATA".S2_oper,
           delta                    := 1,
           proport_o                := "F2_DATA".pzd2);
_00e: NOP   0;
      A     L 20.1;
      A     "F1";
      JNB   _00f;
      CALL  "加减速子程序" (
           proport                  := "F2_DATA".pzd2,
           oper                     := #S2_di_su,
           delta                    := 1,
           proport_o                := "F2_DATA".pzd2);
_00f: NOP   0;
      A     L 20.0;
      AN    "S4_running_order";
      JNB   _010;
      CALL  "加减速子程序" (
           proport                  := "F2_DATA".pzd2,
           oper                     := 0,
           delta                    := 1,
           proport_o                := "F2_DATA".pzd2);
_010: NOP   0;
NETWORK
TITLE =
      AN    "T 50MS";
      =     L 20.0;
      A(;
      A     L 20.0;
      JNB   _011;
      L     "F2_DATA".pzd2;
      ITD;
      T     #TEMP0;
      SET;
      SAVE;
      CLR;
_011: A     BR;
      );
      JNB   _012;
      L     #TEMP0;
      DTR;
      T     #TEMP3;
_012: NOP   0;
      A(;
      A     L 20.0;
      JNB   _013;
      L     #TEMP3;
      L     #TEMP1;
      *R;
      T     #TEMP3;
      AN    OV;
      SAVE;
      CLR;
_013: A     BR;
      );
      JNB   _014;
      L     #TEMP3;
      RND;
      T     MD 84;
_014: NOP   0;
END_FUNCTION

FUNCTION "显示与通讯程序" : VOID	// FC 84
VERSION : 0.1
BEGIN
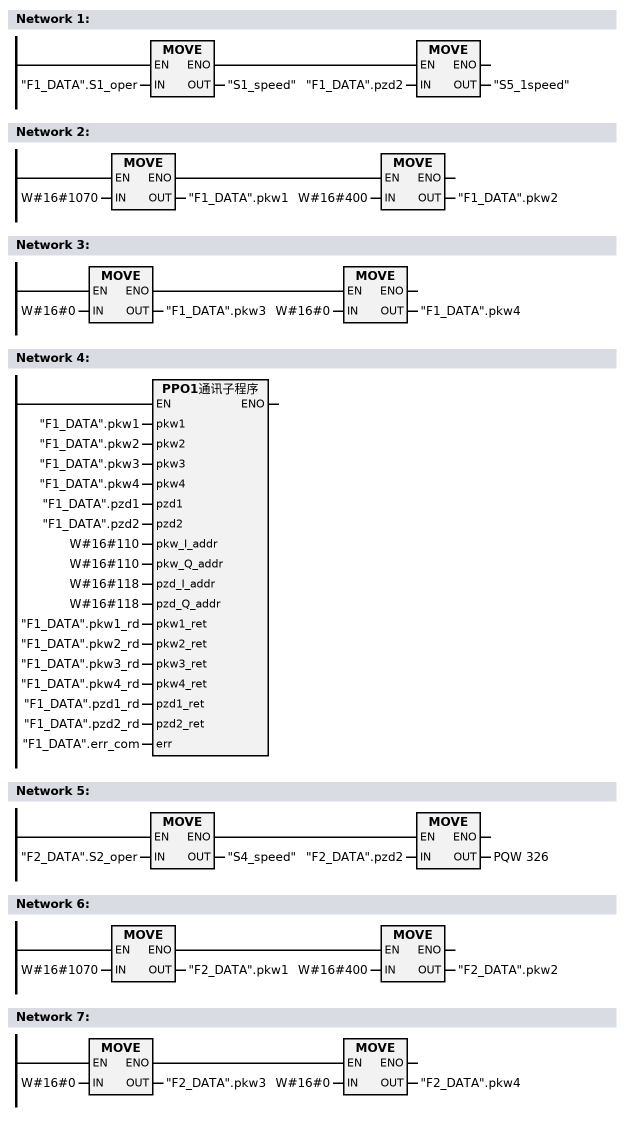
NETWORK
TITLE =
      A(;
      L     "F1_DATA".S1_oper;
      T     "S1_speed";
      SET;
      SAVE;
      CLR;
      A     BR;
      );
      JNB   _001;
      L     "F1_DATA".pzd2;
      T     "S5_1speed";
_001: NOP   0;
NETWORK
TITLE =
      A(;
      L     W#16#1070;
      T     "F1_DATA".pkw1;
      SET;
      SAVE;
      CLR;
      A     BR;
      );
      JNB   _002;
      L     W#16#400;
      T     "F1_DATA".pkw2;
_002: NOP   0;
NETWORK
TITLE =
      A(;
      L     W#16#0;
      T     "F1_DATA".pkw3;
      SET;
      SAVE;
      CLR;
      A     BR;
      );
      JNB   _003;
      L     W#16#0;
      T     "F1_DATA".pkw4;
_003: NOP   0;
NETWORK
TITLE =
      CALL  "PPO1通讯子程序" (
           pkw1                     := "F1_DATA".pkw1,
           pkw2                     := "F1_DATA".pkw2,
           pkw3                     := "F1_DATA".pkw3,
           pkw4                     := "F1_DATA".pkw4,
           pzd1                     := "F1_DATA".pzd1,
           pzd2                     := "F1_DATA".pzd2,
           pkw_I_addr               := W#16#110,
           pkw_Q_addr               := W#16#110,
           pzd_I_addr               := W#16#118,
           pzd_Q_addr               := W#16#118,
           pkw1_ret                 := "F1_DATA".pkw1_rd,
           pkw2_ret                 := "F1_DATA".pkw2_rd,
           pkw3_ret                 := "F1_DATA".pkw3_rd,
           pkw4_ret                 := "F1_DATA".pkw4_rd,
           pzd1_ret                 := "F1_DATA".pzd1_rd,
           pzd2_ret                 := "F1_DATA".pzd2_rd,
           err                      := "F1_DATA".err_com);
      NOP   0;
NETWORK
TITLE =
      A(;
      L     "F2_DATA".S2_oper;
      T     "S4_speed";
      SET;
      SAVE;
      CLR;
      A     BR;
      );
      JNB   _004;
      L     "F2_DATA".pzd2;
      T     PQW 326;
_004: NOP   0;
NETWORK
TITLE =
      A(;
      L     W#16#1070;
      T     "F2_DATA".pkw1;
      SET;
      SAVE;
      CLR;
      A     BR;
      );
      JNB   _005;
      L     W#16#400;
      T     "F2_DATA".pkw2;
_005: NOP   0;
NETWORK
TITLE =
      A(;
      L     W#16#0;
      T     "F2_DATA".pkw3;
      SET;
      SAVE;
      CLR;
      A     BR;
      );
      JNB   _006;
      L     W#16#0;
      T     "F2_DATA".pkw4;
_006: NOP   0;
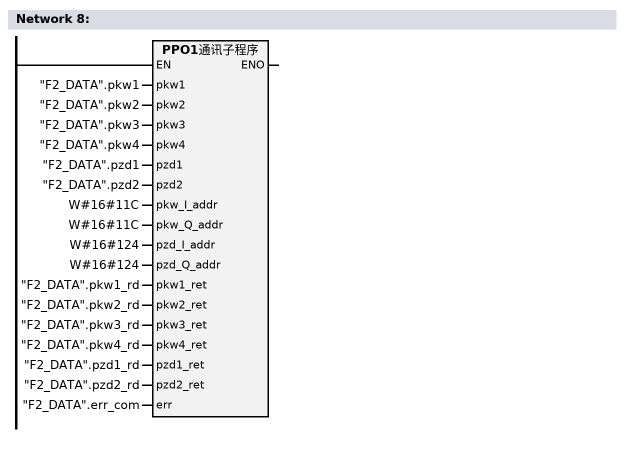
NETWORK
TITLE =
      CALL  "PPO1通讯子程序" (
           pkw1                     := "F2_DATA".pkw1,
           pkw2                     := "F2_DATA".pkw2,
           pkw3                     := "F2_DATA".pkw3,
           pkw4                     := "F2_DATA".pkw4,
           pzd1                     := "F2_DATA".pzd1,
           pzd2                     := "F2_DATA".pzd2,
           pkw_I_addr               := W#16#11C,
           pkw_Q_addr               := W#16#11C,
           pzd_I_addr               := W#16#124,
           pzd_Q_addr               := W#16#124,
           pkw1_ret                 := "F2_DATA".pkw1_rd,
           pkw2_ret                 := "F2_DATA".pkw2_rd,
           pkw3_ret                 := "F2_DATA".pkw3_rd,
           pkw4_ret                 := "F2_DATA".pkw4_rd,
           pzd1_ret                 := "F2_DATA".pzd1_rd,
           pzd2_ret                 := "F2_DATA".pzd2_rd,
           err                      := "F2_DATA".err_com);
      NOP   0;
END_FUNCTION

FUNCTION FC 110 : VOID
VERSION : 0.1
BEGIN
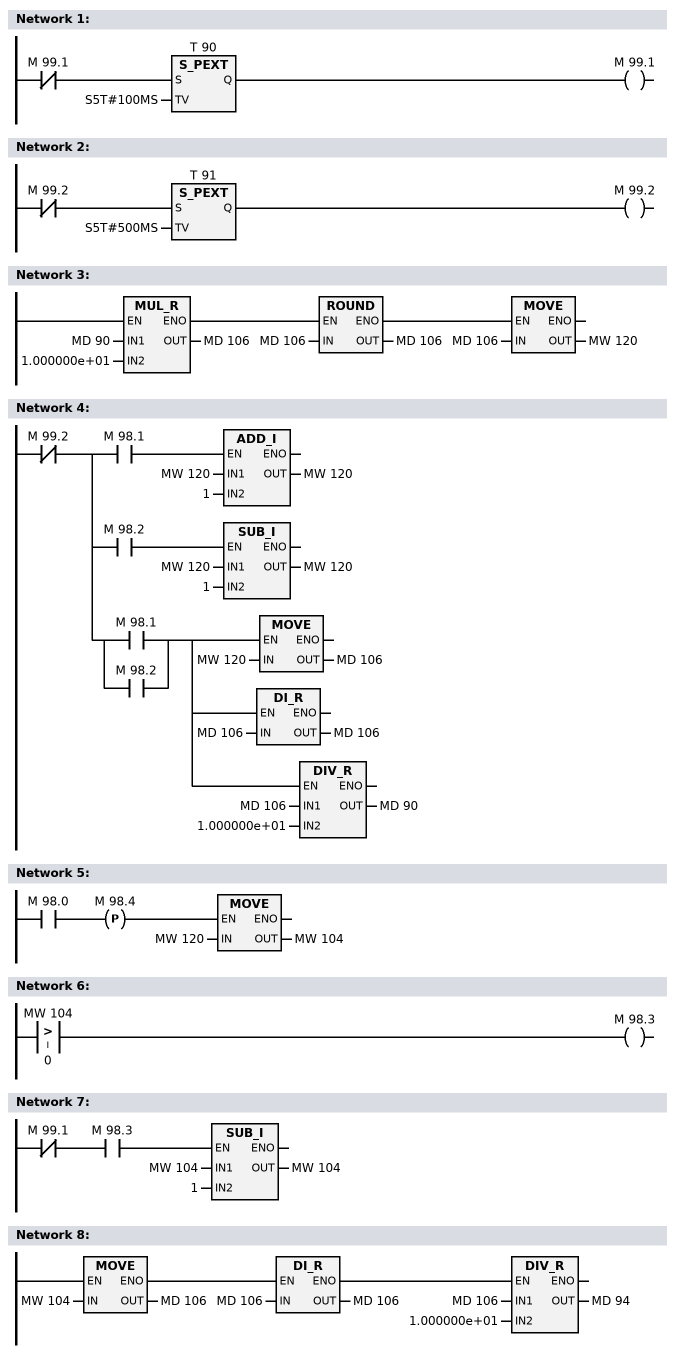
NETWORK
TITLE =
      AN    M 99.1;
      L     S5T#100MS;
      SE    T 90;
      NOP   0;
      NOP   0;
      NOP   0;
      A     T 90;
      =     M 99.1;
NETWORK
TITLE =
      AN    M 99.2;
      L     S5T#500MS;
      SE    T 91;
      NOP   0;
      NOP   0;
      NOP   0;
      A     T 91;
      =     M 99.2;
NETWORK
TITLE =
      A(;
      A(;
      L     MD 90;
      L     1.000000e+01;
      *R;
      T     MD 106;
      AN    OV;
      SAVE;
      CLR;
      A     BR;
      );
      JNB   _001;
      L     MD 106;
      RND;
      T     MD 106;
      AN    OV;
      SAVE;
      CLR;
_001: A     BR;
      );
      JNB   _002;
      L     MD 106;
      T     MW 120;
_002: NOP   0;
NETWORK
TITLE =
      AN    M 99.2;
      =     L 0.0;
      A     L 0.0;
      A     M 98.1;
      JNB   _003;
      L     MW 120;
      L     1;
      +I;
      T     MW 120;
_003: NOP   0;
      A     L 0.0;
      A     M 98.2;
      JNB   _004;
      L     MW 120;
      L     1;
      -I;
      T     MW 120;
_004: NOP   0;
      A     L 0.0;
      A(;
      O     M 98.1;
      O     M 98.2;
      );
      =     L 0.1;
      A     L 0.1;
      JNB   _005;
      L     MW 120;
      T     MD 106;
_005: NOP   0;
      A     L 0.1;
      JNB   _006;
      L     MD 106;
      DTR;
      T     MD 106;
_006: NOP   0;
      A     L 0.1;
      JNB   _007;
      L     MD 106;
      L     1.000000e+01;
      /R;
      T     MD 90;
_007: NOP   0;
NETWORK
TITLE =
      A     M 98.0;
      FP    M 98.4;
      JNB   _008;
      L     MW 120;
      T     MW 104;
_008: NOP   0;
NETWORK
TITLE =
      L     MW 104;
      L     0;
      >I;
      =     M 98.3;
NETWORK
TITLE =
      AN    M 99.1;
      A     M 98.3;
      JNB   _009;
      L     MW 104;
      L     1;
      -I;
      T     MW 104;
_009: NOP   0;
NETWORK
TITLE =
      A(;
      A(;
      L     MW 104;
      T     MD 106;
      SET;
      SAVE;
      CLR;
      A     BR;
      );
      JNB   _00a;
      L     MD 106;
      DTR;
      T     MD 106;
      SET;
      SAVE;
      CLR;
_00a: A     BR;
      );
      JNB   _00b;
      L     MD 106;
      L     1.000000e+01;
      /R;
      T     MD 94;
_00b: NOP   0;
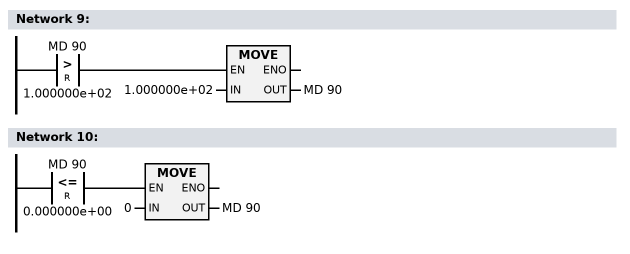
NETWORK
TITLE =
      A(;
      L     MD 90;
      L     1.000000e+02;
      >R;
      );
      JNB   _00c;
      L     1.000000e+02;
      T     MD 90;
_00c: NOP   0;
NETWORK
TITLE =
      A(;
      L     MD 90;
      L     0.000000e+00;
      <=R;
      );
      JNB   _00d;
      L     0;
      T     MD 90;
_00d: NOP   0;
END_FUNCTION

FUNCTION FC 111 : VOID
VERSION : 0.1
BEGIN
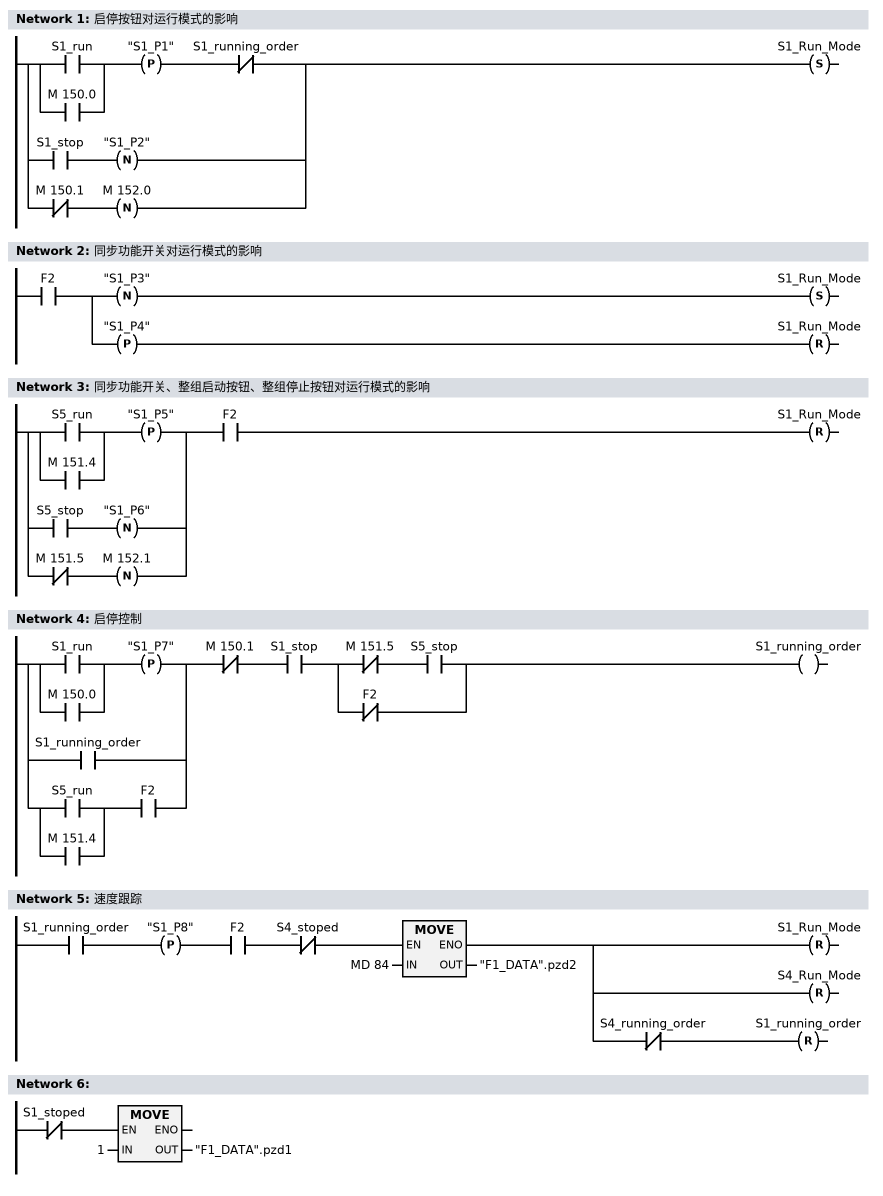
NETWORK
TITLE = 启停按钮对运行模式的影响
//Run_Mode=1表示单机运行，Run_Mode=0表示同步运行
      A(;
      O     "S1_run";
      O     M 150.0;
      );
      FP    "S1_P1";
      AN    "S1_running_order";
      O(;
      A     "S1_stop";
      FN    "S1_P2";
      );
      O(;
      AN    M 150.1;
      FN    M 152.0;
      );
      S     "S1_Run_Mode";
NETWORK
TITLE = 同步功能开关对运行模式的影响
//Run_Mode=1表示单机运行，Run_Mode=0表示同步运行
      A     "F2";
      =     L 0.0;
      A     L 0.0;
      FN    "S1_P3";
      S     "S1_Run_Mode";
      A     L 0.0;
      FP    "S1_P4";
      R     "S1_Run_Mode";
NETWORK
TITLE = 同步功能开关、整组启动按钮、整组停止按钮对运行模式的影响
//Run_Mode=1表示单机运行，Run_Mode=0表示同步运行
//“S3启动”（I1.0）为整组启动按钮，“S3停止”（I1.1）为整组停止按钮。
      A(;
      A(;
      O     "S5_run";
      O     M 151.4;
      );
      FP    "S1_P5";
      O(;
      A     "S5_stop";
      FN    "S1_P6";
      );
      O(;
      AN    M 151.5;
      FN    M 152.1;
      );
      );
      A     "F2";
      R     "S1_Run_Mode";
NETWORK
TITLE = 启停控制
//“F2”（I6.1）为同步功能开关，即I6.1=0时，两台变频器单机运行，I6.1=1时，两台变频
//器同步运行
      A(;
      A(;
      O     "S1_run";
      O     M 150.0;
      );
      FP    "S1_P7";
      O     "S1_running_order";
      O;
      A(;
      O     "S5_run";
      O     M 151.4;
      );
      A     "F2";
      );
      AN    M 150.1;
      A     "S1_stop";
      A(;
      AN    M 151.5;
      A     "S5_stop";
      ON    "F2";
      );
      =     "S1_running_order";
NETWORK
TITLE = 速度跟踪
//Run_Mode=1表示单机运行，Run_Mode=0表示同步运行
      A     "S1_running_order";
      FP    "S1_P8";
      A     "F2";
      AN    "S4_stoped";
      JNB   _001;
      L     MD 84;
      T     "F1_DATA".pzd2;
      SET;
      SAVE;
      CLR;
_001: A     BR;
      =     L 0.0;
      A     L 0.0;
      BLD   102;
      R     "S1_Run_Mode";
      A     L 0.0;
      BLD   102;
      R     "S4_Run_Mode";
      A     L 0.0;
      AN    "S4_running_order";
      R     "S1_running_order";
NETWORK
TITLE =
      AN    "S1_stoped";
      JNB   _002;
      L     1;
      T     "F1_DATA".pzd1;
_002: NOP   0;
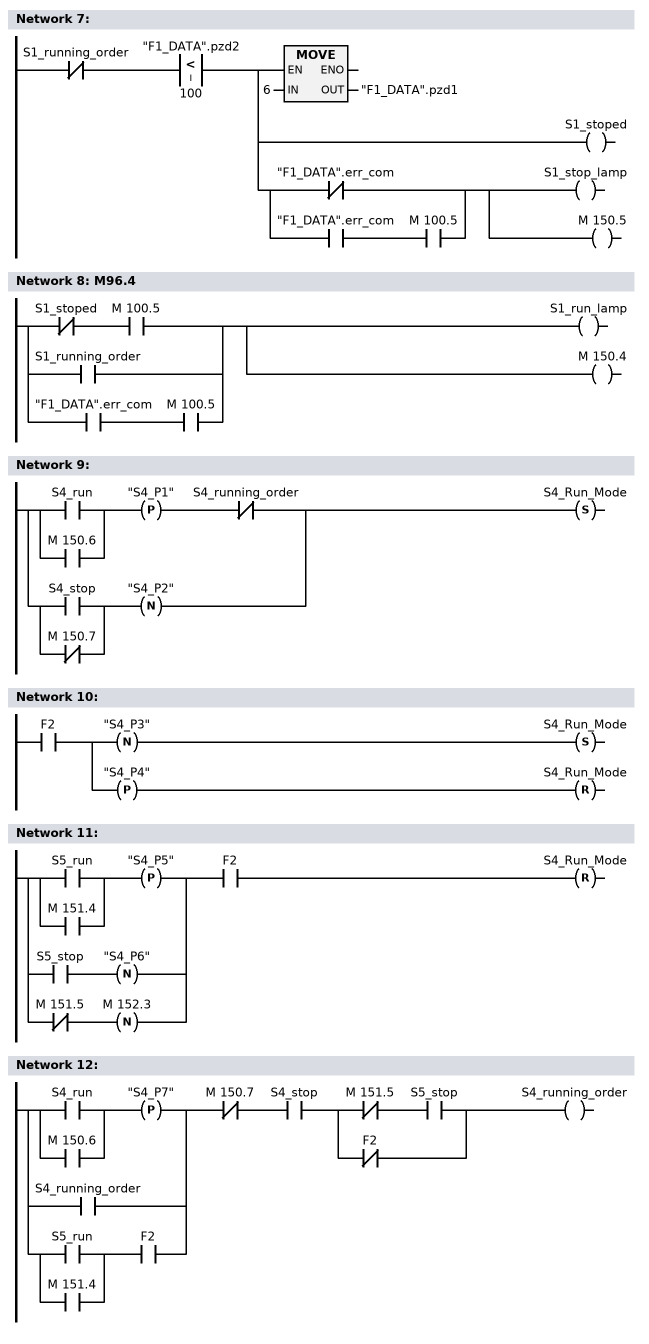
NETWORK
TITLE =
      AN    "S1_running_order";
      A(;
      L     "F1_DATA".pzd2;
      L     100;
      <I;
      );
      =     L 0.0;
      A     L 0.0;
      JNB   _003;
      L     6;
      T     "F1_DATA".pzd1;
_003: NOP   0;
      A     L 0.0;
      BLD   102;
      =     "S1_stoped";
      A     L 0.0;
      A(;
      ON    "F1_DATA".err_com;
      O;
      A     "F1_DATA".err_com;
      A     M 100.5;
      );
      =     "S1_stop_lamp";
      =     M 150.5;
NETWORK
TITLE = M96.4
      AN    "S1_stoped";
      A     M 100.5;
      O     "S1_running_order";
      O;
      A     "F1_DATA".err_com;
      A     M 100.5;
      =     "S1_run_lamp";
      =     M 150.4;
NETWORK
TITLE =
      A(;
      O     "S4_run";
      O     M 150.6;
      );
      FP    "S4_P1";
      AN    "S4_running_order";
      O(;
      A(;
      O     "S4_stop";
      ON    M 150.7;
      );
      FN    "S4_P2";
      );
      S     "S4_Run_Mode";
NETWORK
TITLE =
      A     "F2";
      =     L 0.0;
      A     L 0.0;
      FN    "S4_P3";
      S     "S4_Run_Mode";
      A     L 0.0;
      FP    "S4_P4";
      R     "S4_Run_Mode";
NETWORK
TITLE =
      A(;
      A(;
      O     "S5_run";
      O     M 151.4;
      );
      FP    "S4_P5";
      O(;
      A     "S5_stop";
      FN    "S4_P6";
      );
      O(;
      AN    M 151.5;
      FN    M 152.3;
      );
      );
      A     "F2";
      R     "S4_Run_Mode";
NETWORK
TITLE =
      A(;
      A(;
      O     "S4_run";
      O     M 150.6;
      );
      FP    "S4_P7";
      O     "S4_running_order";
      O;
      A(;
      O     "S5_run";
      O     M 151.4;
      );
      A     "F2";
      );
      AN    M 150.7;
      A     "S4_stop";
      A(;
      AN    M 151.5;
      A     "S5_stop";
      ON    "F2";
      );
      =     "S4_running_order";
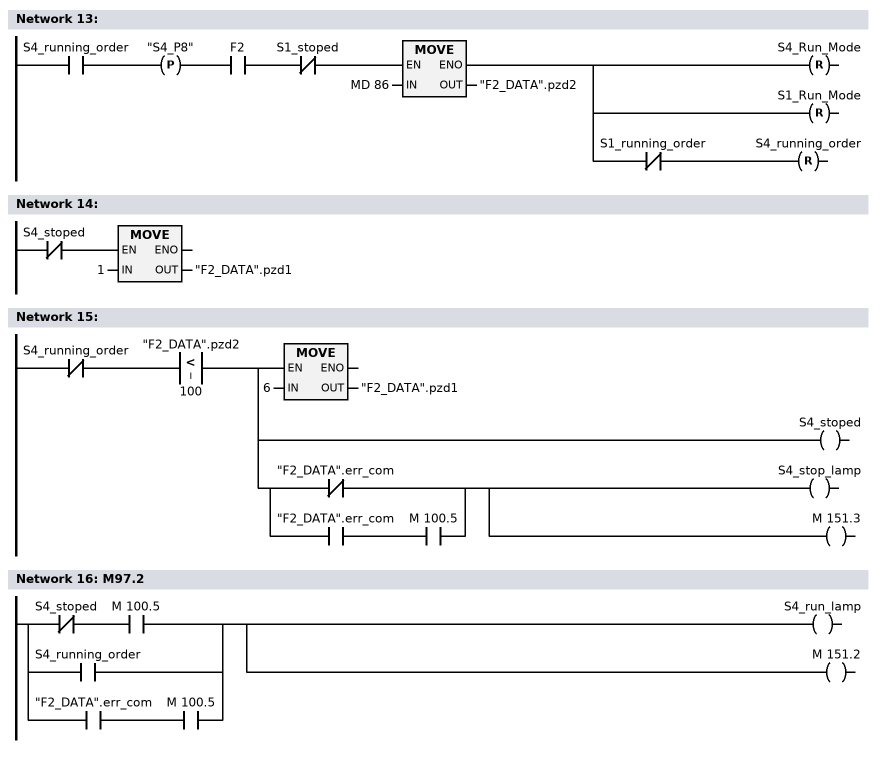
NETWORK
TITLE =
      A     "S4_running_order";
      FP    "S4_P8";
      A     "F2";
      AN    "S1_stoped";
      JNB   _004;
      L     MD 86;
      T     "F2_DATA".pzd2;
      SET;
      SAVE;
      CLR;
_004: A     BR;
      =     L 0.0;
      A     L 0.0;
      BLD   102;
      R     "S4_Run_Mode";
      A     L 0.0;
      BLD   102;
      R     "S1_Run_Mode";
      A     L 0.0;
      AN    "S1_running_order";
      R     "S4_running_order";
NETWORK
TITLE =
      AN    "S4_stoped";
      JNB   _005;
      L     1;
      T     "F2_DATA".pzd1;
_005: NOP   0;
NETWORK
TITLE =
      AN    "S4_running_order";
      A(;
      L     "F2_DATA".pzd2;
      L     100;
      <I;
      );
      =     L 0.0;
      A     L 0.0;
      JNB   _006;
      L     6;
      T     "F2_DATA".pzd1;
_006: NOP   0;
      A     L 0.0;
      BLD   102;
      =     "S4_stoped";
      A     L 0.0;
      A(;
      ON    "F2_DATA".err_com;
      O;
      A     "F2_DATA".err_com;
      A     M 100.5;
      );
      =     "S4_stop_lamp";
      =     M 151.3;
NETWORK
TITLE = M97.2
      AN    "S4_stoped";
      A     M 100.5;
      O     "S4_running_order";
      O;
      A     "F2_DATA".err_com;
      A     M 100.5;
      =     "S4_run_lamp";
      =     M 151.2;
END_FUNCTION

FUNCTION FC 112 : VOID
VERSION : 0.1
VAR_TEMP
  S1_di_su : INT ;
  S2_di_su : INT ;
END_VAR
BEGIN
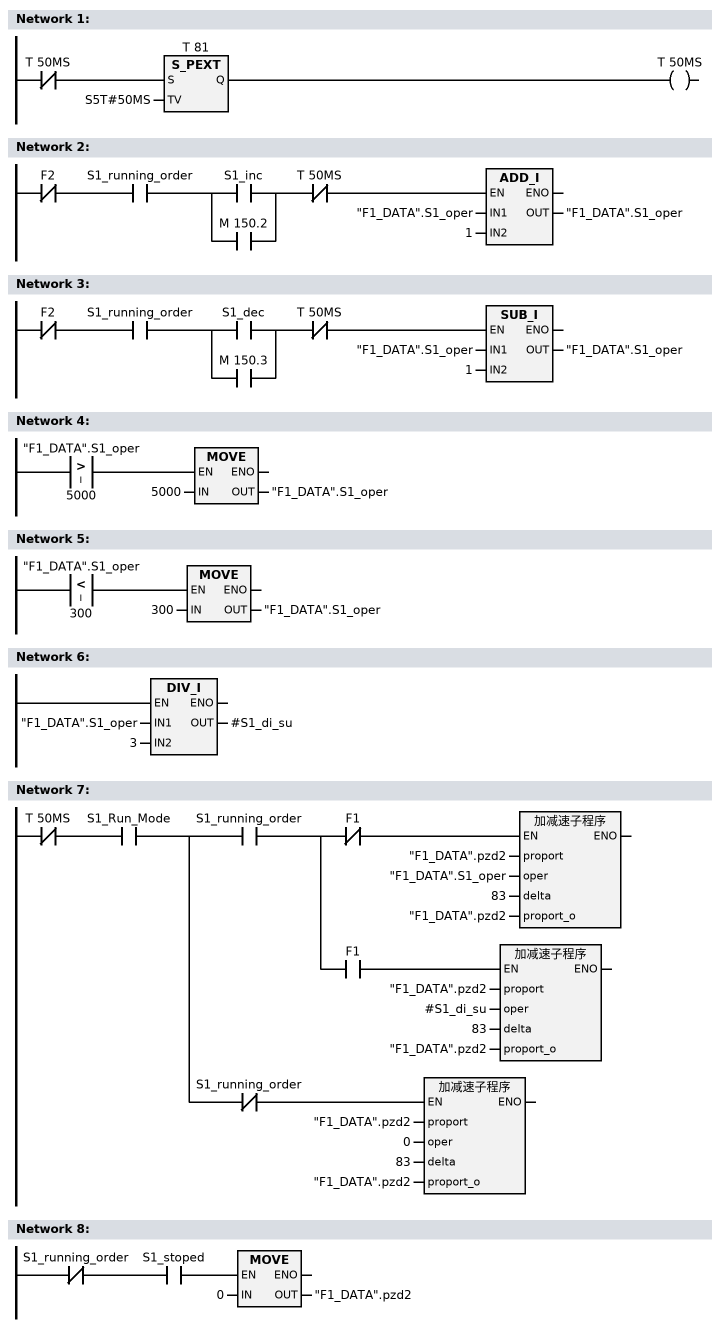
NETWORK
TITLE =
      AN    "T 50MS";
      L     S5T#50MS;
      SE    T 81;
      NOP   0;
      NOP   0;
      NOP   0;
      A     T 81;
      =     "T 50MS";
NETWORK
TITLE =
      AN    "F2";
      A     "S1_running_order";
      A(;
      O     "S1_inc";
      O     M 150.2;
      );
      AN    "T 50MS";
      JNB   _001;
      L     "F1_DATA".S1_oper;
      L     1;
      +I;
      T     "F1_DATA".S1_oper;
_001: NOP   0;
NETWORK
TITLE =
      AN    "F2";
      A     "S1_running_order";
      A(;
      O     "S1_dec";
      O     M 150.3;
      );
      AN    "T 50MS";
      JNB   _002;
      L     "F1_DATA".S1_oper;
      L     1;
      -I;
      T     "F1_DATA".S1_oper;
_002: NOP   0;
NETWORK
TITLE =
      A(;
      L     "F1_DATA".S1_oper;
      L     5000;
      >I;
      );
      JNB   _003;
      L     5000;
      T     "F1_DATA".S1_oper;
_003: NOP   0;
NETWORK
TITLE =
      A(;
      L     "F1_DATA".S1_oper;
      L     300;
      <I;
      );
      JNB   _004;
      L     300;
      T     "F1_DATA".S1_oper;
_004: NOP   0;
NETWORK
TITLE =
      L     "F1_DATA".S1_oper;
      L     3;
      /I;
      T     #S1_di_su;
      NOP   0;
NETWORK
TITLE =
      AN    "T 50MS";
      A     "S1_Run_Mode";
      =     L 4.0;
      A     L 4.0;
      A     "S1_running_order";
      =     L 4.1;
      A     L 4.1;
      AN    "F1";
      JNB   _005;
      CALL  "加减速子程序" (
           proport                  := "F1_DATA".pzd2,
           oper                     := "F1_DATA".S1_oper,
           delta                    := 83,
           proport_o                := "F1_DATA".pzd2);
_005: NOP   0;
      A     L 4.1;
      A     "F1";
      JNB   _006;
      CALL  "加减速子程序" (
           proport                  := "F1_DATA".pzd2,
           oper                     := #S1_di_su,
           delta                    := 83,
           proport_o                := "F1_DATA".pzd2);
_006: NOP   0;
      A     L 4.0;
      AN    "S1_running_order";
      JNB   _007;
      CALL  "加减速子程序" (
           proport                  := "F1_DATA".pzd2,
           oper                     := 0,
           delta                    := 83,
           proport_o                := "F1_DATA".pzd2);
_007: NOP   0;
NETWORK
TITLE =
      AN    "S1_running_order";
      A     "S1_stoped";
      JNB   _008;
      L     0;
      T     "F1_DATA".pzd2;
_008: NOP   0;
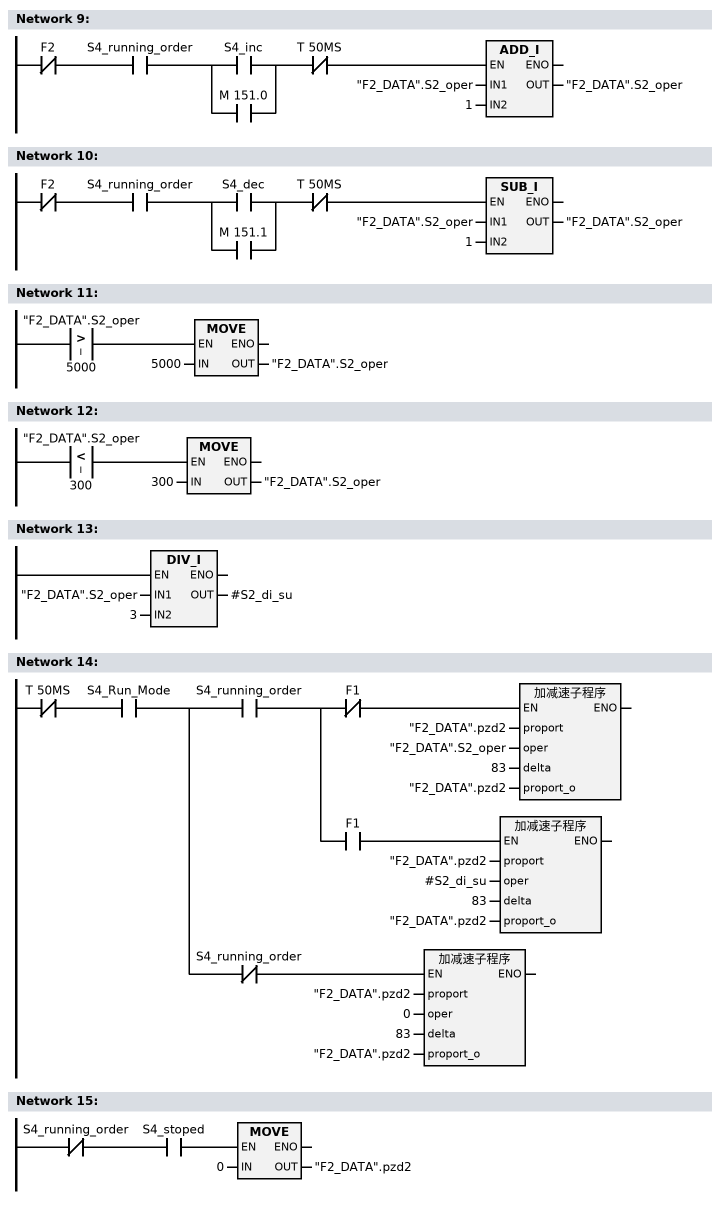
NETWORK
TITLE =
      AN    "F2";
      A     "S4_running_order";
      A(;
      O     "S4_inc";
      O     M 151.0;
      );
      AN    "T 50MS";
      JNB   _009;
      L     "F2_DATA".S2_oper;
      L     1;
      +I;
      T     "F2_DATA".S2_oper;
_009: NOP   0;
NETWORK
TITLE =
      AN    "F2";
      A     "S4_running_order";
      A(;
      O     "S4_dec";
      O     M 151.1;
      );
      AN    "T 50MS";
      JNB   _00a;
      L     "F2_DATA".S2_oper;
      L     1;
      -I;
      T     "F2_DATA".S2_oper;
_00a: NOP   0;
NETWORK
TITLE =
      A(;
      L     "F2_DATA".S2_oper;
      L     5000;
      >I;
      );
      JNB   _00b;
      L     5000;
      T     "F2_DATA".S2_oper;
_00b: NOP   0;
NETWORK
TITLE =
      A(;
      L     "F2_DATA".S2_oper;
      L     300;
      <I;
      );
      JNB   _00c;
      L     300;
      T     "F2_DATA".S2_oper;
_00c: NOP   0;
NETWORK
TITLE =
      L     "F2_DATA".S2_oper;
      L     3;
      /I;
      T     #S2_di_su;
      NOP   0;
NETWORK
TITLE =
      AN    "T 50MS";
      A     "S4_Run_Mode";
      =     L 4.0;
      A     L 4.0;
      A     "S4_running_order";
      =     L 4.1;
      A     L 4.1;
      AN    "F1";
      JNB   _00d;
      CALL  "加减速子程序" (
           proport                  := "F2_DATA".pzd2,
           oper                     := "F2_DATA".S2_oper,
           delta                    := 83,
           proport_o                := "F2_DATA".pzd2);
_00d: NOP   0;
      A     L 4.1;
      A     "F1";
      JNB   _00e;
      CALL  "加减速子程序" (
           proport                  := "F2_DATA".pzd2,
           oper                     := #S2_di_su,
           delta                    := 83,
           proport_o                := "F2_DATA".pzd2);
_00e: NOP   0;
      A     L 4.0;
      AN    "S4_running_order";
      JNB   _00f;
      CALL  "加减速子程序" (
           proport                  := "F2_DATA".pzd2,
           oper                     := 0,
           delta                    := 83,
           proport_o                := "F2_DATA".pzd2);
_00f: NOP   0;
NETWORK
TITLE =
      AN    "S4_running_order";
      A     "S4_stoped";
      JNB   _010;
      L     0;
      T     "F2_DATA".pzd2;
_010: NOP   0;
END_FUNCTION

FUNCTION FC 113 : VOID
VERSION : 0.1
VAR_TEMP
  TEMP0 : DINT ;
  TEMP1 : REAL ;
  TEMP2 : DINT ;
  TEMP3 : REAL ;
  S1_di_su : INT ;
  S2_di_su : INT ;
END_VAR
BEGIN
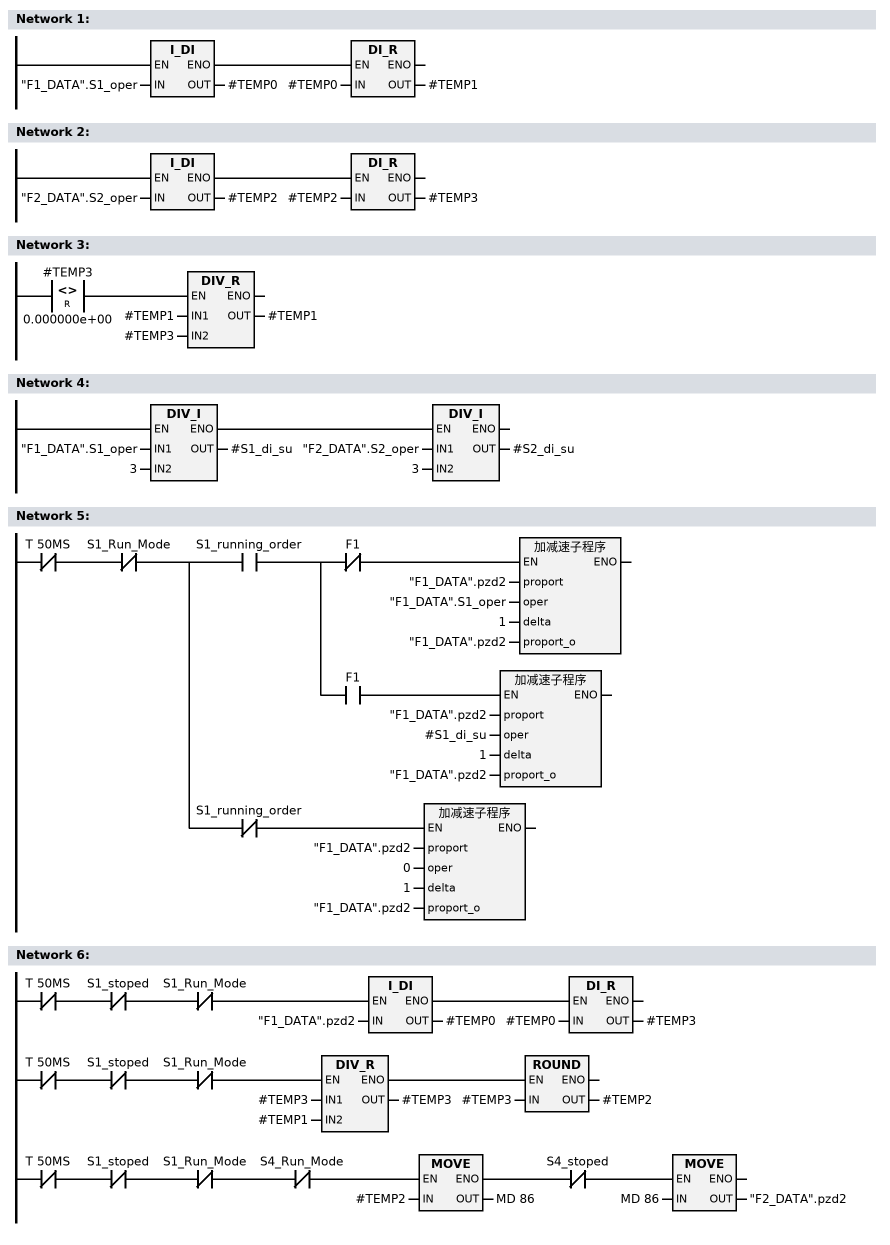
NETWORK
TITLE =
      A(;
      L     "F1_DATA".S1_oper;
      ITD;
      T     #TEMP0;
      SET;
      SAVE;
      CLR;
      A     BR;
      );
      JNB   _001;
      L     #TEMP0;
      DTR;
      T     #TEMP1;
_001: NOP   0;
NETWORK
TITLE =
      A(;
      L     "F2_DATA".S2_oper;
      ITD;
      T     #TEMP2;
      SET;
      SAVE;
      CLR;
      A     BR;
      );
      JNB   _002;
      L     #TEMP2;
      DTR;
      T     #TEMP3;
_002: NOP   0;
NETWORK
TITLE =
      A(;
      L     #TEMP3;
      L     0.000000e+00;
      <>R;
      );
      JNB   _003;
      L     #TEMP1;
      L     #TEMP3;
      /R;
      T     #TEMP1;
_003: NOP   0;
NETWORK
TITLE =
      A(;
      L     "F1_DATA".S1_oper;
      L     3;
      /I;
      T     #S1_di_su;
      AN    OV;
      SAVE;
      CLR;
      A     BR;
      );
      JNB   _004;
      L     "F2_DATA".S2_oper;
      L     3;
      /I;
      T     #S2_di_su;
_004: NOP   0;
NETWORK
TITLE =
      AN    "T 50MS";
      AN    "S1_Run_Mode";
      =     L 20.0;
      A     L 20.0;
      A     "S1_running_order";
      =     L 20.1;
      A     L 20.1;
      AN    "F1";
      JNB   _005;
      CALL  "加减速子程序" (
           proport                  := "F1_DATA".pzd2,
           oper                     := "F1_DATA".S1_oper,
           delta                    := 1,
           proport_o                := "F1_DATA".pzd2);
_005: NOP   0;
      A     L 20.1;
      A     "F1";
      JNB   _006;
      CALL  "加减速子程序" (
           proport                  := "F1_DATA".pzd2,
           oper                     := #S1_di_su,
           delta                    := 1,
           proport_o                := "F1_DATA".pzd2);
_006: NOP   0;
      A     L 20.0;
      AN    "S1_running_order";
      JNB   _007;
      CALL  "加减速子程序" (
           proport                  := "F1_DATA".pzd2,
           oper                     := 0,
           delta                    := 1,
           proport_o                := "F1_DATA".pzd2);
_007: NOP   0;
NETWORK
TITLE =
      AN    "T 50MS";
      AN    "S1_stoped";
      AN    "S1_Run_Mode";
      =     L 20.0;
      A(;
      A     L 20.0;
      JNB   _008;
      L     "F1_DATA".pzd2;
      ITD;
      T     #TEMP0;
      SET;
      SAVE;
      CLR;
_008: A     BR;
      );
      JNB   _009;
      L     #TEMP0;
      DTR;
      T     #TEMP3;
_009: NOP   0;
      A(;
      A     L 20.0;
      JNB   _00a;
      L     #TEMP3;
      L     #TEMP1;
      /R;
      T     #TEMP3;
      AN    OV;
      SAVE;
      CLR;
_00a: A     BR;
      );
      JNB   _00b;
      L     #TEMP3;
      RND;
      T     #TEMP2;
_00b: NOP   0;
      A(;
      A     L 20.0;
      AN    "S4_Run_Mode";
      JNB   _00c;
      L     #TEMP2;
      T     MD 86;
      SET;
      SAVE;
      CLR;
_00c: A     BR;
      );
      AN    "S4_stoped";
      JNB   _00d;
      L     MD 86;
      T     "F2_DATA".pzd2;
_00d: NOP   0;
